DATA_BLOCK "n0016-uc164-xn10_SN50_2"   // DB1008, F_DB
{ S7_Optimized_Access := 'TRUE' }
VERSION : 0.1
// stored: InstanceOfName 00_Push-Button_Input
"00_Push-Button_Input"
BEGIN
END_DATA_BLOCK

DATA_BLOCK "n0020-uc15-el001-k30001_SN50_1"   // DB1009, F_DB
{ S7_Optimized_Access := 'TRUE' }
VERSION : 0.1
// stored: InstanceOfName 00_Push-Button_Input
"00_Push-Button_Input"
BEGIN
END_DATA_BLOCK

DATA_BLOCK "n0020-uc15-el001-k30001_SN50_2"   // DB1010, F_DB
{ S7_Optimized_Access := 'TRUE' }
VERSION : 0.1
// stored: InstanceOfName 00_Push-Button_Input
"00_Push-Button_Input"
BEGIN
END_DATA_BLOCK

DATA_BLOCK "n0020-uc15-el001-k30001_SN50_3"   // DB1011, F_DB
{ S7_Optimized_Access := 'TRUE' }
VERSION : 0.1
// stored: InstanceOfName 00_Push-Button_Input
"00_Push-Button_Input"
BEGIN
END_DATA_BLOCK

DATA_BLOCK "n0023-uc154-xn10_SN50_1"   // DB1012, F_DB
{ S7_Optimized_Access := 'TRUE' }
VERSION : 0.1
// stored: InstanceOfName 00_Push-Button_Input
"00_Push-Button_Input"
BEGIN
END_DATA_BLOCK

DATA_BLOCK "n0023-uc154-xn10_SN50_2"   // DB1013, F_DB
{ S7_Optimized_Access := 'TRUE' }
VERSION : 0.1
// stored: InstanceOfName 00_Push-Button_Input
"00_Push-Button_Input"
BEGIN
END_DATA_BLOCK

DATA_BLOCK "n0021-icg11-el001-k30001_SN50_1"   // DB1014, F_DB
{ S7_Optimized_Access := 'TRUE' }
VERSION : 0.1
// stored: InstanceOfName 00_Push-Button_Input
"00_Push-Button_Input"
BEGIN
END_DATA_BLOCK

DATA_BLOCK "n0021-icg11-el001-k30001_SN50_2"   // DB1015, F_DB
{ S7_Optimized_Access := 'TRUE' }
VERSION : 0.1
// stored: InstanceOfName 00_Push-Button_Input
"00_Push-Button_Input"
BEGIN
END_DATA_BLOCK

DATA_BLOCK "n0021-icg11-el001-k30001_SN50_3"   // DB1016, F_DB
{ S7_Optimized_Access := 'TRUE' }
VERSION : 0.1
// stored: InstanceOfName 00_Push-Button_Input
"00_Push-Button_Input"
BEGIN
END_DATA_BLOCK

DATA_BLOCK "n0021-icg11-el001-k30001_SN50_4"   // DB1017, F_DB
{ S7_Optimized_Access := 'TRUE' }
VERSION : 0.1
// stored: InstanceOfName 00_Push-Button_Input
"00_Push-Button_Input"
BEGIN
END_DATA_BLOCK

DATA_BLOCK "n0022-icg21-el001-k30001_SN50_1"   // DB1018, F_DB
{ S7_Optimized_Access := 'TRUE' }
VERSION : 0.1
// stored: InstanceOfName 00_Push-Button_Input
"00_Push-Button_Input"
BEGIN
END_DATA_BLOCK

DATA_BLOCK "n0022-icg21-el001-k30001_SN50_2"   // DB1019, F_DB
{ S7_Optimized_Access := 'TRUE' }
VERSION : 0.1
// stored: InstanceOfName 00_Push-Button_Input
"00_Push-Button_Input"
BEGIN
END_DATA_BLOCK

DATA_BLOCK "n0025-uc14-el001-k30001_SN50_1"   // DB1020, F_DB
{ S7_Optimized_Access := 'TRUE' }
VERSION : 0.1
// stored: InstanceOfName 00_Push-Button_Input
"00_Push-Button_Input"
BEGIN
END_DATA_BLOCK

DATA_BLOCK "n0025-uc14-el001-k30001_SN50_2"   // DB1021, F_DB
{ S7_Optimized_Access := 'TRUE' }
VERSION : 0.1
// stored: InstanceOfName 00_Push-Button_Input
"00_Push-Button_Input"
BEGIN
END_DATA_BLOCK

DATA_BLOCK "n0025-uc14-el001-k30001_SN50_3"   // DB1022, F_DB
{ S7_Optimized_Access := 'TRUE' }
VERSION : 0.1
// stored: InstanceOfName 00_Push-Button_Input
"00_Push-Button_Input"
BEGIN
END_DATA_BLOCK

DATA_BLOCK "n0026-uc144-xn10_SN50_1"   // DB1023, F_DB
{ S7_Optimized_Access := 'TRUE' }
VERSION : 0.1
// stored: InstanceOfName 00_Push-Button_Input
"00_Push-Button_Input"
BEGIN
END_DATA_BLOCK

DATA_BLOCK "n0026-uc144-xn10_SN50_2"   // DB1024, F_DB
{ S7_Optimized_Access := 'TRUE' }
VERSION : 0.1
// stored: InstanceOfName 00_Push-Button_Input
"00_Push-Button_Input"
BEGIN
END_DATA_BLOCK

DATA_BLOCK "n0038-uc1-el001-k30001_SN50_1"   // DB1025, F_DB
{ S7_Optimized_Access := 'TRUE' }
VERSION : 0.1
// stored: InstanceOfName 00_Push-Button_Input
"00_Push-Button_Input"
BEGIN
END_DATA_BLOCK

DATA_BLOCK "n0041-uf31-el002-k30001_SN50_1"   // DB1026, F_DB
{ S7_Optimized_Access := 'TRUE' }
VERSION : 0.1
// stored: InstanceOfName 00_Push-Button_Input
"00_Push-Button_Input"
BEGIN
END_DATA_BLOCK

DATA_BLOCK "n0044-ct1-el001-k30001_SN50_1"   // DB1027, F_DB
{ S7_Optimized_Access := 'TRUE' }
VERSION : 0.1
// stored: InstanceOfName 00_Push-Button_Input
"00_Push-Button_Input"
BEGIN
END_DATA_BLOCK

DATA_BLOCK "n0044-ct1-el001-k30001_SN50_2"   // DB1028, F_DB
{ S7_Optimized_Access := 'TRUE' }
VERSION : 0.1
// stored: InstanceOfName 00_Push-Button_Input
"00_Push-Button_Input"
BEGIN
END_DATA_BLOCK

DATA_BLOCK "n0044-ct1-el001-k30001_SN50_3"   // DB1029, F_DB
{ S7_Optimized_Access := 'TRUE' }
VERSION : 0.1
// stored: InstanceOfName 00_Push-Button_Input
"00_Push-Button_Input"
BEGIN
END_DATA_BLOCK

DATA_BLOCK "n0044-ct1-el001-k30001_SN50_4"   // DB1030, F_DB
{ S7_Optimized_Access := 'TRUE' }
VERSION : 0.1
// stored: InstanceOfName 00_Push-Button_Input
"00_Push-Button_Input"
BEGIN
END_DATA_BLOCK

DATA_BLOCK "n0045-ct1-el002-k30001_SN50_1"   // DB1031, F_DB
{ S7_Optimized_Access := 'TRUE' }
VERSION : 0.1
// stored: InstanceOfName 00_Push-Button_Input
"00_Push-Button_Input"
BEGIN
END_DATA_BLOCK

DATA_BLOCK "n0045-ct1-el002-k30001_SN50_2"   // DB1032, F_DB
{ S7_Optimized_Access := 'TRUE' }
VERSION : 0.1
// stored: InstanceOfName 00_Push-Button_Input
"00_Push-Button_Input"
BEGIN
END_DATA_BLOCK

DATA_BLOCK "n0045-ct1-el002-k30001_SN50_3"   // DB1033, F_DB
{ S7_Optimized_Access := 'TRUE' }
VERSION : 0.1
// stored: InstanceOfName 00_Push-Button_Input
"00_Push-Button_Input"
BEGIN
END_DATA_BLOCK

DATA_BLOCK "n0045-ct1-el002-k30001_SN50_4"   // DB1034, F_DB
{ S7_Optimized_Access := 'TRUE' }
VERSION : 0.1
// stored: InstanceOfName 00_Push-Button_Input
"00_Push-Button_Input"
BEGIN
END_DATA_BLOCK

DATA_BLOCK "n0045-ct1-el002-k30001_SN50_5"   // DB1035, F_DB
{ S7_Optimized_Access := 'TRUE' }
VERSION : 0.1
// stored: InstanceOfName 00_Push-Button_Input
"00_Push-Button_Input"
BEGIN
END_DATA_BLOCK

DATA_BLOCK "n0046-ct1-el003-k30001_SN50_1"   // DB1036, F_DB
{ S7_Optimized_Access := 'TRUE' }
VERSION : 0.1
// stored: InstanceOfName 00_Push-Button_Input
"00_Push-Button_Input"
BEGIN
END_DATA_BLOCK

DATA_BLOCK "n0046-ct1-el003-k30001_SN50_2"   // DB1037, F_DB
{ S7_Optimized_Access := 'TRUE' }
VERSION : 0.1
// stored: InstanceOfName 00_Push-Button_Input
"00_Push-Button_Input"
BEGIN
END_DATA_BLOCK

DATA_BLOCK "n0046-ct1-el003-k30001_SN50_3"   // DB1038, F_DB
{ S7_Optimized_Access := 'TRUE' }
VERSION : 0.1
// stored: InstanceOfName 00_Push-Button_Input
"00_Push-Button_Input"
BEGIN
END_DATA_BLOCK

DATA_BLOCK "n0046-ct1-el003-k30001_SN50_4"   // DB1039, F_DB
{ S7_Optimized_Access := 'TRUE' }
VERSION : 0.1
// stored: InstanceOfName 00_Push-Button_Input
"00_Push-Button_Input"
BEGIN
END_DATA_BLOCK

DATA_BLOCK "n0050-uc13-el001-k30001_SN50_1"   // DB1040, F_DB
{ S7_Optimized_Access := 'TRUE' }
VERSION : 0.1
// stored: InstanceOfName 00_Push-Button_Input
"00_Push-Button_Input"
BEGIN
END_DATA_BLOCK

DATA_BLOCK "n0050-uc13-el001-k30001_SN50_2"   // DB1041, F_DB
{ S7_Optimized_Access := 'TRUE' }
VERSION : 0.1
// stored: InstanceOfName 00_Push-Button_Input
"00_Push-Button_Input"
BEGIN
END_DATA_BLOCK

DATA_BLOCK "n0050-uc13-el001-k30001_SN50_3"   // DB1042, F_DB
{ S7_Optimized_Access := 'TRUE' }
VERSION : 0.1
// stored: InstanceOfName 00_Push-Button_Input
"00_Push-Button_Input"
BEGIN
END_DATA_BLOCK

DATA_BLOCK "n0051-uc134-xn10_SN50_1"   // DB1043, F_DB
{ S7_Optimized_Access := 'TRUE' }
VERSION : 0.1
// stored: InstanceOfName 00_Push-Button_Input
"00_Push-Button_Input"
BEGIN
END_DATA_BLOCK

DATA_BLOCK "n0051-uc134-xn10_SN50_2"   // DB1044, F_DB
{ S7_Optimized_Access := 'TRUE' }
VERSION : 0.1
// stored: InstanceOfName 00_Push-Button_Input
"00_Push-Button_Input"
BEGIN
END_DATA_BLOCK

DATA_BLOCK "n0053-uc12-el001-k30001_SN50_1"   // DB1045, F_DB
{ S7_Optimized_Access := 'TRUE' }
VERSION : 0.1
// stored: InstanceOfName 00_Push-Button_Input
"00_Push-Button_Input"
BEGIN
END_DATA_BLOCK

DATA_BLOCK "n0053-uc12-el001-k30001_SN50_2"   // DB1046, F_DB
{ S7_Optimized_Access := 'TRUE' }
VERSION : 0.1
// stored: InstanceOfName 00_Push-Button_Input
"00_Push-Button_Input"
BEGIN
END_DATA_BLOCK

DATA_BLOCK "n0053-uc12-el001-k30001_SN50_3"   // DB1047, F_DB
{ S7_Optimized_Access := 'TRUE' }
VERSION : 0.1
// stored: InstanceOfName 00_Push-Button_Input
"00_Push-Button_Input"
BEGIN
END_DATA_BLOCK

DATA_BLOCK "n0055-uc124-xn10_SN50_1"   // DB1048, F_DB
{ S7_Optimized_Access := 'TRUE' }
VERSION : 0.1
// stored: InstanceOfName 00_Push-Button_Input
"00_Push-Button_Input"
BEGIN
END_DATA_BLOCK

DATA_BLOCK "n0055-uc124-xn10_SN50_2"   // DB1049, F_DB
{ S7_Optimized_Access := 'TRUE' }
VERSION : 0.1
// stored: InstanceOfName 00_Push-Button_Input
"00_Push-Button_Input"
BEGIN
END_DATA_BLOCK

DATA_BLOCK "n0057-uc11-el001-k30001_SN50_1"   // DB1050, F_DB
{ S7_Optimized_Access := 'TRUE' }
VERSION : 0.1
// stored: InstanceOfName 00_Push-Button_Input
"00_Push-Button_Input"
BEGIN
END_DATA_BLOCK

DATA_BLOCK "n0057-uc11-el001-k30001_SN50_2"   // DB1051, F_DB
{ S7_Optimized_Access := 'TRUE' }
VERSION : 0.1
// stored: InstanceOfName 00_Push-Button_Input
"00_Push-Button_Input"
BEGIN
END_DATA_BLOCK

DATA_BLOCK "n0057-uc11-el001-k30001_SN50_3"   // DB1052, F_DB
{ S7_Optimized_Access := 'TRUE' }
VERSION : 0.1
// stored: InstanceOfName 00_Push-Button_Input
"00_Push-Button_Input"
BEGIN
END_DATA_BLOCK

DATA_BLOCK "n0060-uc114-xn10_SN50_1"   // DB1053, F_DB
{ S7_Optimized_Access := 'TRUE' }
VERSION : 0.1
// stored: InstanceOfName 00_Push-Button_Input
"00_Push-Button_Input"
BEGIN
END_DATA_BLOCK

DATA_BLOCK "n0060-uc114-xn10_SN50_2"   // DB1054, F_DB
{ S7_Optimized_Access := 'TRUE' }
VERSION : 0.1
// stored: InstanceOfName 00_Push-Button_Input
"00_Push-Button_Input"
BEGIN
END_DATA_BLOCK

DATA_BLOCK "n0028-uc17-el001-k30001_SN50_1"   // DB1055, F_DB
{ S7_Optimized_Access := 'TRUE' }
VERSION : 0.1
// stored: InstanceOfName 00_Push-Button_Input
"00_Push-Button_Input"
BEGIN
END_DATA_BLOCK

DATA_BLOCK "n0028-uc17-el001-k30001_SN50_2"   // DB1056, F_DB
{ S7_Optimized_Access := 'TRUE' }
VERSION : 0.1
// stored: InstanceOfName 00_Push-Button_Input
"00_Push-Button_Input"
BEGIN
END_DATA_BLOCK

DATA_BLOCK "n0029-uc173-xn10_SN50_1"   // DB1057, F_DB
{ S7_Optimized_Access := 'TRUE' }
VERSION : 0.1
// stored: InstanceOfName 00_Push-Button_Input
"00_Push-Button_Input"
BEGIN
END_DATA_BLOCK

DATA_BLOCK "n0029-uc173-xn10_SN50_2"   // DB1058, F_DB
{ S7_Optimized_Access := 'TRUE' }
VERSION : 0.1
// stored: InstanceOfName 00_Push-Button_Input
"00_Push-Button_Input"
BEGIN
END_DATA_BLOCK

DATA_BLOCK "n0033-zp001-el001-k40001_SN50_1"   // DB1059, F_DB
{ S7_Optimized_Access := 'TRUE' }
VERSION : 0.1
// stored: InstanceOfName 00_Push-Button_Input
"00_Push-Button_Input"
BEGIN
END_DATA_BLOCK

DATA_BLOCK "n0033-zp001-el001-k40001_SN50_2"   // DB1060, F_DB
{ S7_Optimized_Access := 'TRUE' }
VERSION : 0.1
// stored: InstanceOfName 00_Push-Button_Input
"00_Push-Button_Input"
BEGIN
END_DATA_BLOCK

DATA_BLOCK "n0033-zp001-el001-k40001_SN50_3"   // DB1061, F_DB
{ S7_Optimized_Access := 'TRUE' }
VERSION : 0.1
// stored: InstanceOfName 00_Push-Button_Input
"00_Push-Button_Input"
BEGIN
END_DATA_BLOCK

DATA_BLOCK "n0034-ug6-el001-k30001_SN50_1"   // DB1062, F_DB
{ S7_Optimized_Access := 'TRUE' }
VERSION : 0.1
// stored: InstanceOfName 00_Push-Button_Input
"00_Push-Button_Input"
BEGIN
END_DATA_BLOCK

DATA_BLOCK "n0034-ug6-el001-k30001_SN50_2"   // DB1063, F_DB
{ S7_Optimized_Access := 'TRUE' }
VERSION : 0.1
// stored: InstanceOfName 00_Push-Button_Input
"00_Push-Button_Input"
BEGIN
END_DATA_BLOCK

DATA_BLOCK "n0034-ug6-el001-k30001_SN50_3"   // DB1064, F_DB
{ S7_Optimized_Access := 'TRUE' }
VERSION : 0.1
// stored: InstanceOfName 00_Push-Button_Input
"00_Push-Button_Input"
BEGIN
END_DATA_BLOCK

DATA_BLOCK "n0035-ug6-xn10_SN50_1"   // DB1065, F_DB
{ S7_Optimized_Access := 'TRUE' }
VERSION : 0.1
// stored: InstanceOfName 00_Push-Button_Input
"00_Push-Button_Input"
BEGIN
END_DATA_BLOCK

DATA_BLOCK "n0035-ug6-xn10_SN50_2"   // DB1066, F_DB
{ S7_Optimized_Access := 'TRUE' }
VERSION : 0.1
// stored: InstanceOfName 00_Push-Button_Input
"00_Push-Button_Input"
BEGIN
END_DATA_BLOCK

DATA_BLOCK "n0043-db93-el001-k30001_SN50_1"   // DB1067, F_DB
{ S7_Optimized_Access := 'TRUE' }
VERSION : 0.1
// stored: InstanceOfName 00_Push-Button_Input
"00_Push-Button_Input"
BEGIN
END_DATA_BLOCK

DATA_BLOCK "n0031-db931-xn10_SN50_1"   // DB1068, F_DB
{ S7_Optimized_Access := 'TRUE' }
VERSION : 0.1
// stored: InstanceOfName 00_Push-Button_Input
"00_Push-Button_Input"
BEGIN
END_DATA_BLOCK

DATA_BLOCK "n0031-db931-xn10_SN50_2"   // DB1069, F_DB
{ S7_Optimized_Access := 'TRUE' }
VERSION : 0.1
// stored: InstanceOfName 00_Push-Button_Input
"00_Push-Button_Input"
BEGIN
END_DATA_BLOCK

DATA_BLOCK "n0005-lv008-el001-k30001_SN51_1"   // DB1070, F_DB
{ S7_Optimized_Access := 'TRUE' }
VERSION : 0.1
// stored: InstanceOfName 00_Push-Button_Input
"00_Push-Button_Input"
BEGIN
END_DATA_BLOCK

DATA_BLOCK "n0006-lv008-el001-k30001_SN51_1"   // DB1071, F_DB
{ S7_Optimized_Access := 'TRUE' }
VERSION : 0.1
// stored: InstanceOfName 00_Push-Button_Input
"00_Push-Button_Input"
BEGIN
END_DATA_BLOCK

DATA_BLOCK "n0007-icg22-el001-k30001_SN51_1"   // DB1072, F_DB
{ S7_Optimized_Access := 'TRUE' }
VERSION : 0.1
// stored: InstanceOfName 00_Push-Button_Input
"00_Push-Button_Input"
BEGIN
END_DATA_BLOCK

DATA_BLOCK "n0007-icg22-el001-k30001_SN51_2"   // DB1073, F_DB
{ S7_Optimized_Access := 'TRUE' }
VERSION : 0.1
// stored: InstanceOfName 00_Push-Button_Input
"00_Push-Button_Input"
BEGIN
END_DATA_BLOCK

DATA_BLOCK "n0008-icg12-el001-k30001_SN51_1"   // DB1074, F_DB
{ S7_Optimized_Access := 'TRUE' }
VERSION : 0.1
// stored: InstanceOfName 00_Push-Button_Input
"00_Push-Button_Input"
BEGIN
END_DATA_BLOCK

DATA_BLOCK "n0008-icg12-el001-k30001_SN51_2"   // DB1075, F_DB
{ S7_Optimized_Access := 'TRUE' }
VERSION : 0.1
// stored: InstanceOfName 00_Push-Button_Input
"00_Push-Button_Input"
BEGIN
END_DATA_BLOCK

DATA_BLOCK "n0008-icg12-el001-k30001_SN51_3"   // DB1076, F_DB
{ S7_Optimized_Access := 'TRUE' }
VERSION : 0.1
// stored: InstanceOfName 00_Push-Button_Input
"00_Push-Button_Input"
BEGIN
END_DATA_BLOCK

DATA_BLOCK "n0008-icg12-el001-k30001_SN51_4"   // DB1077, F_DB
{ S7_Optimized_Access := 'TRUE' }
VERSION : 0.1
// stored: InstanceOfName 00_Push-Button_Input
"00_Push-Button_Input"
BEGIN
END_DATA_BLOCK

DATA_BLOCK "n0026-uc915-xn10_SN51_1"   // DB1078, F_DB
{ S7_Optimized_Access := 'TRUE' }
VERSION : 0.1
// stored: InstanceOfName 00_Push-Button_Input
"00_Push-Button_Input"
BEGIN
END_DATA_BLOCK

DATA_BLOCK "n0026-uc915-xn10_SN51_2"   // DB1079, F_DB
{ S7_Optimized_Access := 'TRUE' }
VERSION : 0.1
// stored: InstanceOfName 00_Push-Button_Input
"00_Push-Button_Input"
BEGIN
END_DATA_BLOCK

DATA_BLOCK "n0027-uc915-xn11_SN51_1"   // DB1080, F_DB
{ S7_Optimized_Access := 'TRUE' }
VERSION : 0.1
// stored: InstanceOfName 00_Push-Button_Input
"00_Push-Button_Input"
BEGIN
END_DATA_BLOCK

DATA_BLOCK "n0029-ct2-el001-k30001_SN51_1"   // DB1081, F_DB
{ S7_Optimized_Access := 'TRUE' }
VERSION : 0.1
// stored: InstanceOfName 00_Push-Button_Input
"00_Push-Button_Input"
BEGIN
END_DATA_BLOCK

DATA_BLOCK "n0029-ct2-el001-k30001_SN51_2"   // DB1082, F_DB
{ S7_Optimized_Access := 'TRUE' }
VERSION : 0.1
// stored: InstanceOfName 00_Push-Button_Input
"00_Push-Button_Input"
BEGIN
END_DATA_BLOCK

DATA_BLOCK "n0029-ct2-el001-k30001_SN51_3"   // DB1083, F_DB
{ S7_Optimized_Access := 'TRUE' }
VERSION : 0.1
// stored: InstanceOfName 00_Push-Button_Input
"00_Push-Button_Input"
BEGIN
END_DATA_BLOCK

DATA_BLOCK "n0029-ct2-el001-k30001_SN51_4"   // DB1084, F_DB
{ S7_Optimized_Access := 'TRUE' }
VERSION : 0.1
// stored: InstanceOfName 00_Push-Button_Input
"00_Push-Button_Input"
BEGIN
END_DATA_BLOCK

DATA_BLOCK "n0029-ct2-el001-k30001_SN51_5"   // DB1085, F_DB
{ S7_Optimized_Access := 'TRUE' }
VERSION : 0.1
// stored: InstanceOfName 00_Push-Button_Input
"00_Push-Button_Input"
BEGIN
END_DATA_BLOCK

DATA_BLOCK "n0033-uc26-el001-k30001_SN51_1"   // DB1086, F_DB
{ S7_Optimized_Access := 'TRUE' }
VERSION : 0.1
// stored: InstanceOfName 00_Push-Button_Input
"00_Push-Button_Input"
BEGIN
END_DATA_BLOCK

DATA_BLOCK "n0033-uc26-el001-k30001_SN51_2"   // DB1087, F_DB
{ S7_Optimized_Access := 'TRUE' }
VERSION : 0.1
// stored: InstanceOfName 00_Push-Button_Input
"00_Push-Button_Input"
BEGIN
END_DATA_BLOCK

DATA_BLOCK "n0033-uc26-el001-k30001_SN51_3"   // DB1088, F_DB
{ S7_Optimized_Access := 'TRUE' }
VERSION : 0.1
// stored: InstanceOfName 00_Push-Button_Input
"00_Push-Button_Input"
BEGIN
END_DATA_BLOCK

DATA_BLOCK "n0034-uc264-xn10_SN51_1"   // DB1089, F_DB
{ S7_Optimized_Access := 'TRUE' }
VERSION : 0.1
// stored: InstanceOfName 00_Push-Button_Input
"00_Push-Button_Input"
BEGIN
END_DATA_BLOCK

DATA_BLOCK "n0034-uc264-xn10_SN51_2"   // DB1090, F_DB
{ S7_Optimized_Access := 'TRUE' }
VERSION : 0.1
// stored: InstanceOfName 00_Push-Button_Input
"00_Push-Button_Input"
BEGIN
END_DATA_BLOCK

DATA_BLOCK "n0035-ct2-el002-k30001_SN51_1"   // DB1091, F_DB
{ S7_Optimized_Access := 'TRUE' }
VERSION : 0.1
// stored: InstanceOfName 00_Push-Button_Input
"00_Push-Button_Input"
BEGIN
END_DATA_BLOCK

DATA_BLOCK "n0035-ct2-el002-k30001_SN51_2"   // DB1092, F_DB
{ S7_Optimized_Access := 'TRUE' }
VERSION : 0.1
// stored: InstanceOfName 00_Push-Button_Input
"00_Push-Button_Input"
BEGIN
END_DATA_BLOCK

DATA_BLOCK "n0035-ct2-el002-k30001_SN51_3"   // DB1093, F_DB
{ S7_Optimized_Access := 'TRUE' }
VERSION : 0.1
// stored: InstanceOfName 00_Push-Button_Input
"00_Push-Button_Input"
BEGIN
END_DATA_BLOCK

DATA_BLOCK "n0035-ct2-el002-k30001_SN51_4"   // DB1094, F_DB
{ S7_Optimized_Access := 'TRUE' }
VERSION : 0.1
// stored: InstanceOfName 00_Push-Button_Input
"00_Push-Button_Input"
BEGIN
END_DATA_BLOCK

DATA_BLOCK "n0035-ct2-el002-k30001_SN51_5"   // DB1095, F_DB
{ S7_Optimized_Access := 'TRUE' }
VERSION : 0.1
// stored: InstanceOfName 00_Push-Button_Input
"00_Push-Button_Input"
BEGIN
END_DATA_BLOCK

DATA_BLOCK "n0041-uc27-el001-k30001_SN51_1"   // DB1096, F_DB
{ S7_Optimized_Access := 'TRUE' }
VERSION : 0.1
// stored: InstanceOfName 00_Push-Button_Input
"00_Push-Button_Input"
BEGIN
END_DATA_BLOCK

DATA_BLOCK "n0041-uc27-el001-k30001_SN51_2"   // DB1097, F_DB
{ S7_Optimized_Access := 'TRUE' }
VERSION : 0.1
// stored: InstanceOfName 00_Push-Button_Input
"00_Push-Button_Input"
BEGIN
END_DATA_BLOCK

DATA_BLOCK "n0042-uc274-xn10_SN51_1"   // DB1098, F_DB
{ S7_Optimized_Access := 'TRUE' }
VERSION : 0.1
// stored: InstanceOfName 00_Push-Button_Input
"00_Push-Button_Input"
BEGIN
END_DATA_BLOCK

DATA_BLOCK "n0042-uc274-xn10_SN51_2"   // DB1099, F_DB
{ S7_Optimized_Access := 'TRUE' }
VERSION : 0.1
// stored: InstanceOfName 00_Push-Button_Input
"00_Push-Button_Input"
BEGIN
END_DATA_BLOCK

DATA_BLOCK "n0046-uc25-el001-k30001_SN51_1"   // DB1100, F_DB
{ S7_Optimized_Access := 'TRUE' }
VERSION : 0.1
// stored: InstanceOfName 00_Push-Button_Input
"00_Push-Button_Input"
BEGIN
END_DATA_BLOCK

DATA_BLOCK "n0046-uc25-el001-k30001_SN51_2"   // DB1101, F_DB
{ S7_Optimized_Access := 'TRUE' }
VERSION : 0.1
// stored: InstanceOfName 00_Push-Button_Input
"00_Push-Button_Input"
BEGIN
END_DATA_BLOCK

DATA_BLOCK "n0046-uc25-el001-k30001_SN51_3"   // DB1102, F_DB
{ S7_Optimized_Access := 'TRUE' }
VERSION : 0.1
// stored: InstanceOfName 00_Push-Button_Input
"00_Push-Button_Input"
BEGIN
END_DATA_BLOCK

DATA_BLOCK "n0047-uc254-xn10_SN51_1"   // DB1103, F_DB
{ S7_Optimized_Access := 'TRUE' }
VERSION : 0.1
// stored: InstanceOfName 00_Push-Button_Input
"00_Push-Button_Input"
BEGIN
END_DATA_BLOCK

DATA_BLOCK "n0047-uc254-xn10_SN51_2"   // DB1104, F_DB
{ S7_Optimized_Access := 'TRUE' }
VERSION : 0.1
// stored: InstanceOfName 00_Push-Button_Input
"00_Push-Button_Input"
BEGIN
END_DATA_BLOCK

DATA_BLOCK "n0051-uc24-el001-k30001_SN51_1"   // DB1105, F_DB
{ S7_Optimized_Access := 'TRUE' }
VERSION : 0.1
// stored: InstanceOfName 00_Push-Button_Input
"00_Push-Button_Input"
BEGIN
END_DATA_BLOCK

DATA_BLOCK "n0051-uc24-el001-k30001_SN51_2"   // DB1106, F_DB
{ S7_Optimized_Access := 'TRUE' }
VERSION : 0.1
// stored: InstanceOfName 00_Push-Button_Input
"00_Push-Button_Input"
BEGIN
END_DATA_BLOCK

DATA_BLOCK "n0051-uc24-el001-k30001_SN51_3"   // DB1107, F_DB
{ S7_Optimized_Access := 'TRUE' }
VERSION : 0.1
// stored: InstanceOfName 00_Push-Button_Input
"00_Push-Button_Input"
BEGIN
END_DATA_BLOCK

DATA_BLOCK "n0052-uc244-xn10_SN51_1"   // DB1108, F_DB
{ S7_Optimized_Access := 'TRUE' }
VERSION : 0.1
// stored: InstanceOfName 00_Push-Button_Input
"00_Push-Button_Input"
BEGIN
END_DATA_BLOCK

DATA_BLOCK "n0052-uc244-xn10_SN51_2"   // DB1109, F_DB
{ S7_Optimized_Access := 'TRUE' }
VERSION : 0.1
// stored: InstanceOfName 00_Push-Button_Input
"00_Push-Button_Input"
BEGIN
END_DATA_BLOCK

DATA_BLOCK "n0056-uc23-el001-k30001_SN51_1"   // DB1110, F_DB
{ S7_Optimized_Access := 'TRUE' }
VERSION : 0.1
// stored: InstanceOfName 00_Push-Button_Input
"00_Push-Button_Input"
BEGIN
END_DATA_BLOCK

DATA_BLOCK "n0056-uc23-el001-k30001_SN51_2"   // DB1111, F_DB
{ S7_Optimized_Access := 'TRUE' }
VERSION : 0.1
// stored: InstanceOfName 00_Push-Button_Input
"00_Push-Button_Input"
BEGIN
END_DATA_BLOCK

DATA_BLOCK "n0056-uc23-el001-k30001_SN51_3"   // DB1112, F_DB
{ S7_Optimized_Access := 'TRUE' }
VERSION : 0.1
// stored: InstanceOfName 00_Push-Button_Input
"00_Push-Button_Input"
BEGIN
END_DATA_BLOCK

DATA_BLOCK "n0057-uc234-xn10_SN51_1"   // DB1113, F_DB
{ S7_Optimized_Access := 'TRUE' }
VERSION : 0.1
// stored: InstanceOfName 00_Push-Button_Input
"00_Push-Button_Input"
BEGIN
END_DATA_BLOCK

DATA_BLOCK "n0057-uc234-xn10_SN51_2"   // DB1114, F_DB
{ S7_Optimized_Access := 'TRUE' }
VERSION : 0.1
// stored: InstanceOfName 00_Push-Button_Input
"00_Push-Button_Input"
BEGIN
END_DATA_BLOCK

DATA_BLOCK "n0058-ct2-el003-k30001_SN51_1"   // DB1115, F_DB
{ S7_Optimized_Access := 'TRUE' }
VERSION : 0.1
// stored: InstanceOfName 00_Push-Button_Input
"00_Push-Button_Input"
BEGIN
END_DATA_BLOCK

DATA_BLOCK "n0058-ct2-el003-k30001_SN51_2"   // DB1116, F_DB
{ S7_Optimized_Access := 'TRUE' }
VERSION : 0.1
// stored: InstanceOfName 00_Push-Button_Input
"00_Push-Button_Input"
BEGIN
END_DATA_BLOCK

DATA_BLOCK "n0058-ct2-el003-k30001_SN51_3"   // DB1117, F_DB
{ S7_Optimized_Access := 'TRUE' }
VERSION : 0.1
// stored: InstanceOfName 00_Push-Button_Input
"00_Push-Button_Input"
BEGIN
END_DATA_BLOCK

DATA_BLOCK "n0058-ct2-el003-k30001_SN51_4"   // DB1118, F_DB
{ S7_Optimized_Access := 'TRUE' }
VERSION : 0.1
// stored: InstanceOfName 00_Push-Button_Input
"00_Push-Button_Input"
BEGIN
END_DATA_BLOCK

DATA_BLOCK "n0058-ct2-el003-k30001_SN51_5"   // DB1119, F_DB
{ S7_Optimized_Access := 'TRUE' }
VERSION : 0.1
// stored: InstanceOfName 00_Push-Button_Input
"00_Push-Button_Input"
BEGIN
END_DATA_BLOCK

DATA_BLOCK "n0061-uc22-el001-k30001_SN51_1"   // DB1120, F_DB
{ S7_Optimized_Access := 'TRUE' }
VERSION : 0.1
// stored: InstanceOfName 00_Push-Button_Input
"00_Push-Button_Input"
BEGIN
END_DATA_BLOCK

DATA_BLOCK "n0061-uc22-el001-k30001_SN51_2"   // DB1121, F_DB
{ S7_Optimized_Access := 'TRUE' }
VERSION : 0.1
// stored: InstanceOfName 00_Push-Button_Input
"00_Push-Button_Input"
BEGIN
END_DATA_BLOCK

DATA_BLOCK "n0061-uc22-el001-k30001_SN51_3"   // DB1122, F_DB
{ S7_Optimized_Access := 'TRUE' }
VERSION : 0.1
// stored: InstanceOfName 00_Push-Button_Input
"00_Push-Button_Input"
BEGIN
END_DATA_BLOCK

DATA_BLOCK "n0061-uc22-el001-k30001_SN51_4"   // DB1123, F_DB
{ S7_Optimized_Access := 'TRUE' }
VERSION : 0.1
// stored: InstanceOfName 00_Push-Button_Input
"00_Push-Button_Input"
BEGIN
END_DATA_BLOCK

DATA_BLOCK "n0057-uc224-xn10_SN51_1"   // DB1124, F_DB
{ S7_Optimized_Access := 'TRUE' }
VERSION : 0.1
// stored: InstanceOfName 00_Push-Button_Input
"00_Push-Button_Input"
BEGIN
END_DATA_BLOCK

DATA_BLOCK "n0057-uc224-xn10_SN51_2"   // DB1125, F_DB
{ S7_Optimized_Access := 'TRUE' }
VERSION : 0.1
// stored: InstanceOfName 00_Push-Button_Input
"00_Push-Button_Input"
BEGIN
END_DATA_BLOCK

DATA_BLOCK "n0066-uc21-el001-k30001_SN51_1"   // DB1126, F_DB
{ S7_Optimized_Access := 'TRUE' }
VERSION : 0.1
// stored: InstanceOfName 00_Push-Button_Input
"00_Push-Button_Input"
BEGIN
END_DATA_BLOCK

DATA_BLOCK "n0066-uc21-el001-k30001_SN51_2"   // DB1127, F_DB
{ S7_Optimized_Access := 'TRUE' }
VERSION : 0.1
// stored: InstanceOfName 00_Push-Button_Input
"00_Push-Button_Input"
BEGIN
END_DATA_BLOCK

DATA_BLOCK "n0066-uc21-el001-k30001_SN51_3"   // DB1128, F_DB
{ S7_Optimized_Access := 'TRUE' }
VERSION : 0.1
// stored: InstanceOfName 00_Push-Button_Input
"00_Push-Button_Input"
BEGIN
END_DATA_BLOCK

DATA_BLOCK "n0067-uc214-xn10_SN51_1"   // DB1129, F_DB
{ S7_Optimized_Access := 'TRUE' }
VERSION : 0.1
// stored: InstanceOfName 00_Push-Button_Input
"00_Push-Button_Input"
BEGIN
END_DATA_BLOCK

DATA_BLOCK "n0067-uc214-xn10_SN51_2"   // DB1130, F_DB
{ S7_Optimized_Access := 'TRUE' }
VERSION : 0.1
// stored: InstanceOfName 00_Push-Button_Input
"00_Push-Button_Input"
BEGIN
END_DATA_BLOCK

DATA_BLOCK "n0070-uf31-el001-k30001_SN51_1"   // DB1131, F_DB
{ S7_Optimized_Access := 'TRUE' }
VERSION : 0.1
// stored: InstanceOfName 00_Push-Button_Input
"00_Push-Button_Input"
BEGIN
END_DATA_BLOCK

DATA_BLOCK "n0072-uf51-el001-k30001_SN51_1"   // DB1132, F_DB
{ S7_Optimized_Access := 'TRUE' }
VERSION : 0.1
// stored: InstanceOfName 00_Push-Button_Input
"00_Push-Button_Input"
BEGIN
END_DATA_BLOCK

DATA_BLOCK "n0080-uf511-xn10_SN51_1"   // DB1133, F_DB
{ S7_Optimized_Access := 'TRUE' }
VERSION : 0.1
// stored: InstanceOfName 00_Push-Button_Input
"00_Push-Button_Input"
BEGIN
END_DATA_BLOCK

DATA_BLOCK "n0073-ifg31-el001-k30001_SN51_1"   // DB1134, F_DB
{ S7_Optimized_Access := 'TRUE' }
VERSION : 0.1
// stored: InstanceOfName 00_Push-Button_Input
"00_Push-Button_Input"
BEGIN
END_DATA_BLOCK

DATA_BLOCK "n0073-ifg31-el001-k30001_SN51_2"   // DB1135, F_DB
{ S7_Optimized_Access := 'TRUE' }
VERSION : 0.1
// stored: InstanceOfName 00_Push-Button_Input
"00_Push-Button_Input"
BEGIN
END_DATA_BLOCK

DATA_BLOCK "n0074-ifg41-el001-k30001_SN51_1"   // DB1136, F_DB
{ S7_Optimized_Access := 'TRUE' }
VERSION : 0.1
// stored: InstanceOfName 00_Push-Button_Input
"00_Push-Button_Input"
BEGIN
END_DATA_BLOCK

DATA_BLOCK "n0075-uf32-el001-k30001_SN51_1"   // DB1137, F_DB
{ S7_Optimized_Access := 'TRUE' }
VERSION : 0.1
// stored: InstanceOfName 00_Push-Button_Input
"00_Push-Button_Input"
BEGIN
END_DATA_BLOCK

DATA_BLOCK "n0082-zp002-el001-k30001_SN51_1"   // DB1138, F_DB
{ S7_Optimized_Access := 'TRUE' }
VERSION : 0.1
// stored: InstanceOfName 00_Push-Button_Input
"00_Push-Button_Input"
BEGIN
END_DATA_BLOCK

DATA_BLOCK "n0083-lv001-el001-k30001_SN51_1"   // DB1139, F_DB
{ S7_Optimized_Access := 'TRUE' }
VERSION : 0.1
// stored: InstanceOfName 00_Push-Button_Input
"00_Push-Button_Input"
BEGIN
END_DATA_BLOCK

DATA_BLOCK "n0084-lv001-el001-k30001_SN51_1"   // DB1140, F_DB
{ S7_Optimized_Access := 'TRUE' }
VERSION : 0.1
// stored: InstanceOfName 00_Push-Button_Input
"00_Push-Button_Input"
BEGIN
END_DATA_BLOCK

DATA_BLOCK "n0085-uc29-el001-k30001_SN51_1"   // DB1141, F_DB
{ S7_Optimized_Access := 'TRUE' }
VERSION : 0.1
// stored: InstanceOfName 00_Push-Button_Input
"00_Push-Button_Input"
BEGIN
END_DATA_BLOCK

DATA_BLOCK "n0085-uc29-el001-k30001_SN51_2"   // DB1142, F_DB
{ S7_Optimized_Access := 'TRUE' }
VERSION : 0.1
// stored: InstanceOfName 00_Push-Button_Input
"00_Push-Button_Input"
BEGIN
END_DATA_BLOCK

DATA_BLOCK "n0091-zp001-el001-k30001_SN51_1"   // DB1143, F_DB
{ S7_Optimized_Access := 'TRUE' }
VERSION : 0.1
// stored: InstanceOfName 00_Push-Button_Input
"00_Push-Button_Input"
BEGIN
END_DATA_BLOCK

DATA_BLOCK "n0091-zp001-el001-k30001_SN51_2"   // DB1144, F_DB
{ S7_Optimized_Access := 'TRUE' }
VERSION : 0.1
// stored: InstanceOfName 00_Push-Button_Input
"00_Push-Button_Input"
BEGIN
END_DATA_BLOCK

DATA_BLOCK "n0093-ug7-el001-k30001_SN51_1"   // DB1145, F_DB
{ S7_Optimized_Access := 'TRUE' }
VERSION : 0.1
// stored: InstanceOfName 00_Push-Button_Input
"00_Push-Button_Input"
BEGIN
END_DATA_BLOCK

DATA_BLOCK "n0093-ug7-el001-k30001_SN51_2"   // DB1146, F_DB
{ S7_Optimized_Access := 'TRUE' }
VERSION : 0.1
// stored: InstanceOfName 00_Push-Button_Input
"00_Push-Button_Input"
BEGIN
END_DATA_BLOCK

DATA_BLOCK "n0093-ug7-el001-k30001_SN51_3"   // DB1147, F_DB
{ S7_Optimized_Access := 'TRUE' }
VERSION : 0.1
// stored: InstanceOfName 00_Push-Button_Input
"00_Push-Button_Input"
BEGIN
END_DATA_BLOCK

DATA_BLOCK "n0094-ug7-xn10_SN51_1"   // DB1148, F_DB
{ S7_Optimized_Access := 'TRUE' }
VERSION : 0.1
// stored: InstanceOfName 00_Push-Button_Input
"00_Push-Button_Input"
BEGIN
END_DATA_BLOCK

DATA_BLOCK "n0094-ug7-xn10_SN51_2"   // DB1149, F_DB
{ S7_Optimized_Access := 'TRUE' }
VERSION : 0.1
// stored: InstanceOfName 00_Push-Button_Input
"00_Push-Button_Input"
BEGIN
END_DATA_BLOCK

// folder: 01_Feedback error

DATA_BLOCK "FDBACK error_EXAMPLE"   // DB16, F_DB
{ S7_Optimized_Access := 'TRUE' }
VERSION : 0.1
// stored: InstanceOfName 03_FDBACK error
"03_FDBACK error"
BEGIN
END_DATA_BLOCK

DATA_BLOCK "FDBACK-N0001-1"   // DB19, F_DB
{ S7_Optimized_Access := 'TRUE' }
VERSION : 0.1
// stored: InstanceOfName 03_FDBACK error
"03_FDBACK error"
BEGIN
END_DATA_BLOCK

DATA_BLOCK "FDBK_Error_n0015-uc16-el001-k30001_SN50_1"   // DB2000, F_DB
{ S7_Optimized_Access := 'TRUE' }
VERSION : 0.1
// stored: InstanceOfName 03_FDBACK error
"03_FDBACK error"
BEGIN
END_DATA_BLOCK

DATA_BLOCK "FDBK_Error_n0015-uc16-el001-k30001_SN50_2"   // DB2001, F_DB
{ S7_Optimized_Access := 'TRUE' }
VERSION : 0.1
// stored: InstanceOfName 03_FDBACK error
"03_FDBACK error"
BEGIN
END_DATA_BLOCK

DATA_BLOCK "FDBK_Error_n0015-uc16-el001-k30001_SN50_3"   // DB2002, F_DB
{ S7_Optimized_Access := 'TRUE' }
VERSION : 0.1
// stored: InstanceOfName 03_FDBACK error
"03_FDBACK error"
BEGIN
END_DATA_BLOCK

DATA_BLOCK "FDBK_Error_n0017-lv004-el001-k30001_SN50_1"   // DB2003, F_DB
{ S7_Optimized_Access := 'TRUE' }
VERSION : 0.1
// stored: InstanceOfName 03_FDBACK error
"03_FDBACK error"
BEGIN
END_DATA_BLOCK

DATA_BLOCK "FDBK_Error_n0018-lv004-el001-k30001_SN50_1"   // DB2004, F_DB
{ S7_Optimized_Access := 'TRUE' }
VERSION : 0.1
// stored: InstanceOfName 03_FDBACK error
"03_FDBACK error"
BEGIN
END_DATA_BLOCK

DATA_BLOCK "FDBK_Error_n0020-uc15-el001-k30001_SN50_1"   // DB2005, F_DB
{ S7_Optimized_Access := 'TRUE' }
VERSION : 0.1
// stored: InstanceOfName 03_FDBACK error
"03_FDBACK error"
BEGIN
END_DATA_BLOCK

DATA_BLOCK "FDBK_Error_n0020-uc15-el001-k30001_SN50_2"   // DB2006, F_DB
{ S7_Optimized_Access := 'TRUE' }
VERSION : 0.1
// stored: InstanceOfName 03_FDBACK error
"03_FDBACK error"
BEGIN
END_DATA_BLOCK

DATA_BLOCK "FDBK_Error_n0020-uc15-el001-k30001_SN50_3"   // DB2007, F_DB
{ S7_Optimized_Access := 'TRUE' }
VERSION : 0.1
// stored: InstanceOfName 03_FDBACK error
"03_FDBACK error"
BEGIN
END_DATA_BLOCK

DATA_BLOCK "FDBK_Error_n0021-icg11-el001-k30001_SN50_1"   // DB2008, F_DB
{ S7_Optimized_Access := 'TRUE' }
VERSION : 0.1
// stored: InstanceOfName 03_FDBACK error
"03_FDBACK error"
BEGIN
END_DATA_BLOCK

DATA_BLOCK "FDBK_Error_n0022-icg21-el001-k30001_SN50_1"   // DB2009, F_DB
{ S7_Optimized_Access := 'TRUE' }
VERSION : 0.1
// stored: InstanceOfName 03_FDBACK error
"03_FDBACK error"
BEGIN
END_DATA_BLOCK

DATA_BLOCK "FDBK_Error_n0025-uc14-el001-k30001_SN50_1"   // DB2010, F_DB
{ S7_Optimized_Access := 'TRUE' }
VERSION : 0.1
// stored: InstanceOfName 03_FDBACK error
"03_FDBACK error"
BEGIN
END_DATA_BLOCK

DATA_BLOCK "FDBK_Error_n0025-uc14-el001-k30001_SN50_2"   // DB2011, F_DB
{ S7_Optimized_Access := 'TRUE' }
VERSION : 0.1
// stored: InstanceOfName 03_FDBACK error
"03_FDBACK error"
BEGIN
END_DATA_BLOCK

DATA_BLOCK "FDBK_Error_n0025-uc14-el001-k30001_SN50_3"   // DB2012, F_DB
{ S7_Optimized_Access := 'TRUE' }
VERSION : 0.1
// stored: InstanceOfName 03_FDBACK error
"03_FDBACK error"
BEGIN
END_DATA_BLOCK

DATA_BLOCK "FDBK_Error_n0039-lv001-el001-k30001_SN50_1"   // DB2013, F_DB
{ S7_Optimized_Access := 'TRUE' }
VERSION : 0.1
// stored: InstanceOfName 03_FDBACK error
"03_FDBACK error"
BEGIN
END_DATA_BLOCK

DATA_BLOCK "FDBK_Error_n0040-lv001-el001-k30001_SN50_1"   // DB2014, F_DB
{ S7_Optimized_Access := 'TRUE' }
VERSION : 0.1
// stored: InstanceOfName 03_FDBACK error
"03_FDBACK error"
BEGIN
END_DATA_BLOCK

DATA_BLOCK "FDBK_Error_n0041-uf31-el002-k30001_SN50_1"   // DB2015, F_DB
{ S7_Optimized_Access := 'TRUE' }
VERSION : 0.1
// stored: InstanceOfName 03_FDBACK error
"03_FDBACK error"
BEGIN
END_DATA_BLOCK

DATA_BLOCK "FDBK_Error_n0042-uf41-el002-k30001_SN50_1"   // DB2016, F_DB
{ S7_Optimized_Access := 'TRUE' }
VERSION : 0.1
// stored: InstanceOfName 03_FDBACK error
"03_FDBACK error"
BEGIN
END_DATA_BLOCK

DATA_BLOCK "FDBK_Error_n0044-ct1-el001-k30001_SN50_1"   // DB2017, F_DB
{ S7_Optimized_Access := 'TRUE' }
VERSION : 0.1
// stored: InstanceOfName 03_FDBACK error
"03_FDBACK error"
BEGIN
END_DATA_BLOCK

DATA_BLOCK "FDBK_Error_n0045-ct1-el002-k30001_SN50_1"   // DB2018, F_DB
{ S7_Optimized_Access := 'TRUE' }
VERSION : 0.1
// stored: InstanceOfName 03_FDBACK error
"03_FDBACK error"
BEGIN
END_DATA_BLOCK

DATA_BLOCK "FDBK_Error_n0046-ct1-el003-k30001_SN50_1"   // DB2019, F_DB
{ S7_Optimized_Access := 'TRUE' }
VERSION : 0.1
// stored: InstanceOfName 03_FDBACK error
"03_FDBACK error"
BEGIN
END_DATA_BLOCK

DATA_BLOCK "FDBK_Error_n0047-lv002-el001-k30001_SN50_1"   // DB2020, F_DB
{ S7_Optimized_Access := 'TRUE' }
VERSION : 0.1
// stored: InstanceOfName 03_FDBACK error
"03_FDBACK error"
BEGIN
END_DATA_BLOCK

DATA_BLOCK "FDBK_Error_n0048-lv002-el001-k30001_SN50_1"   // DB2021, F_DB
{ S7_Optimized_Access := 'TRUE' }
VERSION : 0.1
// stored: InstanceOfName 03_FDBACK error
"03_FDBACK error"
BEGIN
END_DATA_BLOCK

DATA_BLOCK "FDBK_Error_n0050-uc13-el001-k30001_SN50_1"   // DB2022, F_DB
{ S7_Optimized_Access := 'TRUE' }
VERSION : 0.1
// stored: InstanceOfName 03_FDBACK error
"03_FDBACK error"
BEGIN
END_DATA_BLOCK

DATA_BLOCK "FDBK_Error_n0050-uc13-el001-k30001_SN50_2"   // DB2023, F_DB
{ S7_Optimized_Access := 'TRUE' }
VERSION : 0.1
// stored: InstanceOfName 03_FDBACK error
"03_FDBACK error"
BEGIN
END_DATA_BLOCK

DATA_BLOCK "FDBK_Error_n0050-uc13-el001-k30001_SN50_3"   // DB2024, F_DB
{ S7_Optimized_Access := 'TRUE' }
VERSION : 0.1
// stored: InstanceOfName 03_FDBACK error
"03_FDBACK error"
BEGIN
END_DATA_BLOCK

DATA_BLOCK "FDBK_Error_n0053-uc12-el001-k30001_SN50_1"   // DB2025, F_DB
{ S7_Optimized_Access := 'TRUE' }
VERSION : 0.1
// stored: InstanceOfName 03_FDBACK error
"03_FDBACK error"
BEGIN
END_DATA_BLOCK

DATA_BLOCK "FDBK_Error_n0053-uc12-el001-k30001_SN50_2"   // DB2026, F_DB
{ S7_Optimized_Access := 'TRUE' }
VERSION : 0.1
// stored: InstanceOfName 03_FDBACK error
"03_FDBACK error"
BEGIN
END_DATA_BLOCK

DATA_BLOCK "FDBK_Error_n0053-uc12-el001-k30001_SN50_3"   // DB2027, F_DB
{ S7_Optimized_Access := 'TRUE' }
VERSION : 0.1
// stored: InstanceOfName 03_FDBACK error
"03_FDBACK error"
BEGIN
END_DATA_BLOCK

DATA_BLOCK "FDBK_Error_n0054-uf31-el003-k30001_SN50_1"   // DB2028, F_DB
{ S7_Optimized_Access := 'TRUE' }
VERSION : 0.1
// stored: InstanceOfName 03_FDBACK error
"03_FDBACK error"
BEGIN
END_DATA_BLOCK

DATA_BLOCK "FDBK_Error_n0057-uc11-el001-k30001_SN50_1"   // DB2029, F_DB
{ S7_Optimized_Access := 'TRUE' }
VERSION : 0.1
// stored: InstanceOfName 03_FDBACK error
"03_FDBACK error"
BEGIN
END_DATA_BLOCK

DATA_BLOCK "FDBK_Error_n0057-uc11-el001-k30001_SN50_2"   // DB2030, F_DB
{ S7_Optimized_Access := 'TRUE' }
VERSION : 0.1
// stored: InstanceOfName 03_FDBACK error
"03_FDBACK error"
BEGIN
END_DATA_BLOCK

DATA_BLOCK "FDBK_Error_n0057-uc11-el001-k30001_SN50_3"   // DB2031, F_DB
{ S7_Optimized_Access := 'TRUE' }
VERSION : 0.1
// stored: InstanceOfName 03_FDBACK error
"03_FDBACK error"
BEGIN
END_DATA_BLOCK

DATA_BLOCK "FDBK_Error_n0058-lv003-el001-k30001_SN50_1"   // DB2032, F_DB
{ S7_Optimized_Access := 'TRUE' }
VERSION : 0.1
// stored: InstanceOfName 03_FDBACK error
"03_FDBACK error"
BEGIN
END_DATA_BLOCK

DATA_BLOCK "FDBK_Error_n0059-lv003-el001-k30001_SN50_1"   // DB2033, F_DB
{ S7_Optimized_Access := 'TRUE' }
VERSION : 0.1
// stored: InstanceOfName 03_FDBACK error
"03_FDBACK error"
BEGIN
END_DATA_BLOCK

DATA_BLOCK "FDBK_Error_n0028-uc17-el001-k30001_SN50_1"   // DB2034, F_DB
{ S7_Optimized_Access := 'TRUE' }
VERSION : 0.1
// stored: InstanceOfName 03_FDBACK error
"03_FDBACK error"
BEGIN
END_DATA_BLOCK

DATA_BLOCK "FDBK_Error_n0028-uc17-el001-k30001_SN50_2"   // DB2035, F_DB
{ S7_Optimized_Access := 'TRUE' }
VERSION : 0.1
// stored: InstanceOfName 03_FDBACK error
"03_FDBACK error"
BEGIN
END_DATA_BLOCK

DATA_BLOCK "FDBK_Error_n0033-zp001-el001-k40001_SN50_1"   // DB2036, F_DB
{ S7_Optimized_Access := 'TRUE' }
VERSION : 0.1
// stored: InstanceOfName 03_FDBACK error
"03_FDBACK error"
BEGIN
END_DATA_BLOCK

DATA_BLOCK "FDBK_Error_n0033-zp001-el001-k40001_SN50_2"   // DB2037, F_DB
{ S7_Optimized_Access := 'TRUE' }
VERSION : 0.1
// stored: InstanceOfName 03_FDBACK error
"03_FDBACK error"
BEGIN
END_DATA_BLOCK

DATA_BLOCK "FDBK_Error_n0034-ug6-el001-k30001_SN50_1"   // DB2038, F_DB
{ S7_Optimized_Access := 'TRUE' }
VERSION : 0.1
// stored: InstanceOfName 03_FDBACK error
"03_FDBACK error"
BEGIN
END_DATA_BLOCK

DATA_BLOCK "FDBK_Error_n0034-ug6-el001-k30001_SN50_2"   // DB2039, F_DB
{ S7_Optimized_Access := 'TRUE' }
VERSION : 0.1
// stored: InstanceOfName 03_FDBACK error
"03_FDBACK error"
BEGIN
END_DATA_BLOCK

DATA_BLOCK "FDBK_Error_n0034-ug6-el001-k30001_SN50_3"   // DB2040, F_DB
{ S7_Optimized_Access := 'TRUE' }
VERSION : 0.1
// stored: InstanceOfName 03_FDBACK error
"03_FDBACK error"
BEGIN
END_DATA_BLOCK

DATA_BLOCK "FDBK_Error_n0043-db93-el001-k30001_SN50_1"   // DB2041, F_DB
{ S7_Optimized_Access := 'TRUE' }
VERSION : 0.1
// stored: InstanceOfName 03_FDBACK error
"03_FDBACK error"
BEGIN
END_DATA_BLOCK

DATA_BLOCK "FDBK_Error_n0005-lv008-el001-k30001_SN51_1"   // DB2042, F_DB
{ S7_Optimized_Access := 'TRUE' }
VERSION : 0.1
// stored: InstanceOfName 03_FDBACK error
"03_FDBACK error"
BEGIN
END_DATA_BLOCK

DATA_BLOCK "FDBK_Error_n0006-lv008-el001-k30001_SN51_1"   // DB2043, F_DB
{ S7_Optimized_Access := 'TRUE' }
VERSION : 0.1
// stored: InstanceOfName 03_FDBACK error
"03_FDBACK error"
BEGIN
END_DATA_BLOCK

DATA_BLOCK "FDBK_Error_n0007-icg22-el001-k30001_SN51_1"   // DB2044, F_DB
{ S7_Optimized_Access := 'TRUE' }
VERSION : 0.1
// stored: InstanceOfName 03_FDBACK error
"03_FDBACK error"
BEGIN
END_DATA_BLOCK

DATA_BLOCK "FDBK_Error_n0008-icg12-el001-k30001_SN51_1"   // DB2045, F_DB
{ S7_Optimized_Access := 'TRUE' }
VERSION : 0.1
// stored: InstanceOfName 03_FDBACK error
"03_FDBACK error"
BEGIN
END_DATA_BLOCK

DATA_BLOCK "FDBK_Error_n0009-uf42-el002-k30001_SN51_1"   // DB2046, F_DB
{ S7_Optimized_Access := 'TRUE' }
VERSION : 0.1
// stored: InstanceOfName 03_FDBACK error
"03_FDBACK error"
BEGIN
END_DATA_BLOCK

DATA_BLOCK "FDBK_Error_n0010-lv007-el001-k30001_SN51_1"   // DB2047, F_DB
{ S7_Optimized_Access := 'TRUE' }
VERSION : 0.1
// stored: InstanceOfName 03_FDBACK error
"03_FDBACK error"
BEGIN
END_DATA_BLOCK

DATA_BLOCK "FDBK_Error_n0011-lv007-el001-k30001_SN51_1"   // DB2048, F_DB
{ S7_Optimized_Access := 'TRUE' }
VERSION : 0.1
// stored: InstanceOfName 03_FDBACK error
"03_FDBACK error"
BEGIN
END_DATA_BLOCK

DATA_BLOCK "FDBK_Error_n0025-dc91-el001-k30001_SN51_1"   // DB2049, F_DB
{ S7_Optimized_Access := 'TRUE' }
VERSION : 0.1
// stored: InstanceOfName 03_FDBACK error
"03_FDBACK error"
BEGIN
END_DATA_BLOCK

DATA_BLOCK "FDBK_Error_n0028-lv005-el001-k30001_SN51_1"   // DB2050, F_DB
{ S7_Optimized_Access := 'TRUE' }
VERSION : 0.1
// stored: InstanceOfName 03_FDBACK error
"03_FDBACK error"
BEGIN
END_DATA_BLOCK

DATA_BLOCK "FDBK_Error_n0029-ct2-el001-k30001_SN51_1"   // DB2051, F_DB
{ S7_Optimized_Access := 'TRUE' }
VERSION : 0.1
// stored: InstanceOfName 03_FDBACK error
"03_FDBACK error"
BEGIN
END_DATA_BLOCK

DATA_BLOCK "FDBK_Error_n0033-uc26-el001-k30001_SN51_1"   // DB2052, F_DB
{ S7_Optimized_Access := 'TRUE' }
VERSION : 0.1
// stored: InstanceOfName 03_FDBACK error
"03_FDBACK error"
BEGIN
END_DATA_BLOCK

DATA_BLOCK "FDBK_Error_n0033-uc26-el001-k30001_SN51_2"   // DB2053, F_DB
{ S7_Optimized_Access := 'TRUE' }
VERSION : 0.1
// stored: InstanceOfName 03_FDBACK error
"03_FDBACK error"
BEGIN
END_DATA_BLOCK

DATA_BLOCK "FDBK_Error_n0033-uc26-el001-k30001_SN51_3"   // DB2054, F_DB
{ S7_Optimized_Access := 'TRUE' }
VERSION : 0.1
// stored: InstanceOfName 03_FDBACK error
"03_FDBACK error"
BEGIN
END_DATA_BLOCK

DATA_BLOCK "FDBK_Error_n0035-ct2-el002-k30001_SN51_1"   // DB2055, F_DB
{ S7_Optimized_Access := 'TRUE' }
VERSION : 0.1
// stored: InstanceOfName 03_FDBACK error
"03_FDBACK error"
BEGIN
END_DATA_BLOCK

DATA_BLOCK "FDBK_Error_n0036-lv005-el001-k30001_SN51_1"   // DB2056, F_DB
{ S7_Optimized_Access := 'TRUE' }
VERSION : 0.1
// stored: InstanceOfName 03_FDBACK error
"03_FDBACK error"
BEGIN
END_DATA_BLOCK

DATA_BLOCK "FDBK_Error_n0041-uc27-el001-k30001_SN51_1"   // DB2057, F_DB
{ S7_Optimized_Access := 'TRUE' }
VERSION : 0.1
// stored: InstanceOfName 03_FDBACK error
"03_FDBACK error"
BEGIN
END_DATA_BLOCK

DATA_BLOCK "FDBK_Error_n0041-uc27-el001-k30001_SN51_2"   // DB2058, F_DB
{ S7_Optimized_Access := 'TRUE' }
VERSION : 0.1
// stored: InstanceOfName 03_FDBACK error
"03_FDBACK error"
BEGIN
END_DATA_BLOCK

DATA_BLOCK "FDBK_Error_n0046-uc25-el001-k30001_SN51_1"   // DB2059, F_DB
{ S7_Optimized_Access := 'TRUE' }
VERSION : 0.1
// stored: InstanceOfName 03_FDBACK error
"03_FDBACK error"
BEGIN
END_DATA_BLOCK

DATA_BLOCK "FDBK_Error_n0046-uc25-el001-k30001_SN51_2"   // DB2060, F_DB
{ S7_Optimized_Access := 'TRUE' }
VERSION : 0.1
// stored: InstanceOfName 03_FDBACK error
"03_FDBACK error"
BEGIN
END_DATA_BLOCK

DATA_BLOCK "FDBK_Error_n0046-uc25-el001-k30001_SN51_3"   // DB2061, F_DB
{ S7_Optimized_Access := 'TRUE' }
VERSION : 0.1
// stored: InstanceOfName 03_FDBACK error
"03_FDBACK error"
BEGIN
END_DATA_BLOCK

DATA_BLOCK "FDBK_Error_n0048-lv006-el001-k30001_SN51_1"   // DB2062, F_DB
{ S7_Optimized_Access := 'TRUE' }
VERSION : 0.1
// stored: InstanceOfName 03_FDBACK error
"03_FDBACK error"
BEGIN
END_DATA_BLOCK

DATA_BLOCK "FDBK_Error_n0051-uc24-el001-k30001_SN51_1"   // DB2063, F_DB
{ S7_Optimized_Access := 'TRUE' }
VERSION : 0.1
// stored: InstanceOfName 03_FDBACK error
"03_FDBACK error"
BEGIN
END_DATA_BLOCK

DATA_BLOCK "FDBK_Error_n0051-uc24-el001-k30001_SN51_2"   // DB2064, F_DB
{ S7_Optimized_Access := 'TRUE' }
VERSION : 0.1
// stored: InstanceOfName 03_FDBACK error
"03_FDBACK error"
BEGIN
END_DATA_BLOCK

DATA_BLOCK "FDBK_Error_n0051-uc24-el001-k30001_SN51_3"   // DB2065, F_DB
{ S7_Optimized_Access := 'TRUE' }
VERSION : 0.1
// stored: InstanceOfName 03_FDBACK error
"03_FDBACK error"
BEGIN
END_DATA_BLOCK

DATA_BLOCK "FDBK_Error_n0056-uc23-el001-k30001_SN51_1"   // DB2066, F_DB
{ S7_Optimized_Access := 'TRUE' }
VERSION : 0.1
// stored: InstanceOfName 03_FDBACK error
"03_FDBACK error"
BEGIN
END_DATA_BLOCK

DATA_BLOCK "FDBK_Error_n0056-uc23-el001-k30001_SN51_2"   // DB2067, F_DB
{ S7_Optimized_Access := 'TRUE' }
VERSION : 0.1
// stored: InstanceOfName 03_FDBACK error
"03_FDBACK error"
BEGIN
END_DATA_BLOCK

DATA_BLOCK "FDBK_Error_n0056-uc23-el001-k30001_SN51_3"   // DB2068, F_DB
{ S7_Optimized_Access := 'TRUE' }
VERSION : 0.1
// stored: InstanceOfName 03_FDBACK error
"03_FDBACK error"
BEGIN
END_DATA_BLOCK

DATA_BLOCK "FDBK_Error_n0058-ct2-el003-k30001_SN51_1"   // DB2069, F_DB
{ S7_Optimized_Access := 'TRUE' }
VERSION : 0.1
// stored: InstanceOfName 03_FDBACK error
"03_FDBACK error"
BEGIN
END_DATA_BLOCK

DATA_BLOCK "FDBK_Error_n0061-uc22-el001-k30001_SN51_1"   // DB2070, F_DB
{ S7_Optimized_Access := 'TRUE' }
VERSION : 0.1
// stored: InstanceOfName 03_FDBACK error
"03_FDBACK error"
BEGIN
END_DATA_BLOCK

DATA_BLOCK "FDBK_Error_n0061-uc22-el001-k30001_SN51_2"   // DB2071, F_DB
{ S7_Optimized_Access := 'TRUE' }
VERSION : 0.1
// stored: InstanceOfName 03_FDBACK error
"03_FDBACK error"
BEGIN
END_DATA_BLOCK

DATA_BLOCK "FDBK_Error_n0061-uc22-el001-k30001_SN51_3"   // DB2072, F_DB
{ S7_Optimized_Access := 'TRUE' }
VERSION : 0.1
// stored: InstanceOfName 03_FDBACK error
"03_FDBACK error"
BEGIN
END_DATA_BLOCK

DATA_BLOCK "FDBK_Error_n0063-lv006-el001-k30001_SN51_1"   // DB2073, F_DB
{ S7_Optimized_Access := 'TRUE' }
VERSION : 0.1
// stored: InstanceOfName 03_FDBACK error
"03_FDBACK error"
BEGIN
END_DATA_BLOCK

DATA_BLOCK "FDBK_Error_n0066-uc21-el001-k30001_SN51_1"   // DB2074, F_DB
{ S7_Optimized_Access := 'TRUE' }
VERSION : 0.1
// stored: InstanceOfName 03_FDBACK error
"03_FDBACK error"
BEGIN
END_DATA_BLOCK

DATA_BLOCK "FDBK_Error_n0066-uc21-el001-k30001_SN51_2"   // DB2075, F_DB
{ S7_Optimized_Access := 'TRUE' }
VERSION : 0.1
// stored: InstanceOfName 03_FDBACK error
"03_FDBACK error"
BEGIN
END_DATA_BLOCK

DATA_BLOCK "FDBK_Error_n0066-uc21-el001-k30001_SN51_3"   // DB2076, F_DB
{ S7_Optimized_Access := 'TRUE' }
VERSION : 0.1
// stored: InstanceOfName 03_FDBACK error
"03_FDBACK error"
BEGIN
END_DATA_BLOCK

DATA_BLOCK "FDBK_Error_n0070-uf31-el001-k30001_SN51_1"   // DB2077, F_DB
{ S7_Optimized_Access := 'TRUE' }
VERSION : 0.1
// stored: InstanceOfName 03_FDBACK error
"03_FDBACK error"
BEGIN
END_DATA_BLOCK

DATA_BLOCK "FDBK_Error_n0071-uf41-el001-k30001_SN51_1"   // DB2078, F_DB
{ S7_Optimized_Access := 'TRUE' }
VERSION : 0.1
// stored: InstanceOfName 03_FDBACK error
"03_FDBACK error"
BEGIN
END_DATA_BLOCK

DATA_BLOCK "FDBK_Error_n0072-uf51-el001-k30001_SN51_1"   // DB2079, F_DB
{ S7_Optimized_Access := 'TRUE' }
VERSION : 0.1
// stored: InstanceOfName 03_FDBACK error
"03_FDBACK error"
BEGIN
END_DATA_BLOCK

DATA_BLOCK "FDBK_Error_n0073-ifg31-el001-k30001_SN51_1"   // DB2080, F_DB
{ S7_Optimized_Access := 'TRUE' }
VERSION : 0.1
// stored: InstanceOfName 03_FDBACK error
"03_FDBACK error"
BEGIN
END_DATA_BLOCK

DATA_BLOCK "FDBK_Error_n0074-ifg41-el001-k30001_SN51_1"   // DB2081, F_DB
{ S7_Optimized_Access := 'TRUE' }
VERSION : 0.1
// stored: InstanceOfName 03_FDBACK error
"03_FDBACK error"
BEGIN
END_DATA_BLOCK

DATA_BLOCK "FDBK_Error_n0075-uf32-el001-k30001_SN51_1"   // DB2082, F_DB
{ S7_Optimized_Access := 'TRUE' }
VERSION : 0.1
// stored: InstanceOfName 03_FDBACK error
"03_FDBACK error"
BEGIN
END_DATA_BLOCK

DATA_BLOCK "FDBK_Error_n0076-uf42-el001-k30001_SN51_1"   // DB2083, F_DB
{ S7_Optimized_Access := 'TRUE' }
VERSION : 0.1
// stored: InstanceOfName 03_FDBACK error
"03_FDBACK error"
BEGIN
END_DATA_BLOCK

DATA_BLOCK "FDBK_Error_n0082-zp002-el001-k30001_SN51_1"   // DB2084, F_DB
{ S7_Optimized_Access := 'TRUE' }
VERSION : 0.1
// stored: InstanceOfName 03_FDBACK error
"03_FDBACK error"
BEGIN
END_DATA_BLOCK

DATA_BLOCK "FDBK_Error_n0083-lv001-el001-k30001_SN51_1"   // DB2085, F_DB
{ S7_Optimized_Access := 'TRUE' }
VERSION : 0.1
// stored: InstanceOfName 03_FDBACK error
"03_FDBACK error"
BEGIN
END_DATA_BLOCK

DATA_BLOCK "FDBK_Error_n0084-lv001-el001-k30001_SN51_1"   // DB2086, F_DB
{ S7_Optimized_Access := 'TRUE' }
VERSION : 0.1
// stored: InstanceOfName 03_FDBACK error
"03_FDBACK error"
BEGIN
END_DATA_BLOCK

DATA_BLOCK "FDBK_Error_n0085-uc29-el001-k30001_SN51_1"   // DB2087, F_DB
{ S7_Optimized_Access := 'TRUE' }
VERSION : 0.1
// stored: InstanceOfName 03_FDBACK error
"03_FDBACK error"
BEGIN
END_DATA_BLOCK

DATA_BLOCK "FDBK_Error_n0091-zp001-el001-k30001_SN51_1"   // DB2088, F_DB
{ S7_Optimized_Access := 'TRUE' }
VERSION : 0.1
// stored: InstanceOfName 03_FDBACK error
"03_FDBACK error"
BEGIN
END_DATA_BLOCK

DATA_BLOCK "FDBK_Error_n0091-zp001-el001-k30001_SN51_2"   // DB2089, F_DB
{ S7_Optimized_Access := 'TRUE' }
VERSION : 0.1
// stored: InstanceOfName 03_FDBACK error
"03_FDBACK error"
BEGIN
END_DATA_BLOCK

DATA_BLOCK "FDBK_Error_n0093-ug7-el001-k30001_SN51_1"   // DB2090, F_DB
{ S7_Optimized_Access := 'TRUE' }
VERSION : 0.1
// stored: InstanceOfName 03_FDBACK error
"03_FDBACK error"
BEGIN
END_DATA_BLOCK

DATA_BLOCK "FDBK_Error_n0093-ug7-el001-k30001_SN51_2"   // DB2091, F_DB
{ S7_Optimized_Access := 'TRUE' }
VERSION : 0.1
// stored: InstanceOfName 03_FDBACK error
"03_FDBACK error"
BEGIN
END_DATA_BLOCK

DATA_BLOCK "FDBK_Error_n0093-ug7-el001-k30001_SN51_3"   // DB2092, F_DB
{ S7_Optimized_Access := 'TRUE' }
VERSION : 0.1
// stored: InstanceOfName 03_FDBACK error
"03_FDBACK error"
BEGIN
END_DATA_BLOCK

// folder: 02_Speed Control

DATA_BLOCK "Speed_Control_DB"   // DB17, F_DB
{ S7_Optimized_Access := 'TRUE' }
VERSION : 0.1
// stored: InstanceOfName 01_Speed_Control
"01_Speed_Control"
BEGIN
END_DATA_BLOCK

// folder: 03_Gate manager

DATA_BLOCK "MAINT_DOOR1"   // DB21, F_DB
{ S7_Optimized_Access := 'TRUE' }
VERSION : 0.1
// stored: InstanceOfName 02_Safety_Door
"02_Safety_Door"
BEGIN
END_DATA_BLOCK

// folder: (top level)

FUNCTION_BLOCK "Main_Safety_RTG1"   // FB1, F_FBD
{ S7_Optimized_Access := 'TRUE' }
   VAR_TEMP
      t_Reset : Bool;
   END_VAR
   VAR_TEMP   // added for the SCL form of the ladder/FBD networks
      _w1 : Bool;
      _w2 : Bool;
      _w3 : Bool;
      _w4 : Bool;
      _w5 : Bool;
      _w6 : Bool;
      _w7 : Bool;
      _w8 : Bool;
      _w9 : Bool;
   END_VAR
BEGIN

REGION Network 1: For commissioning
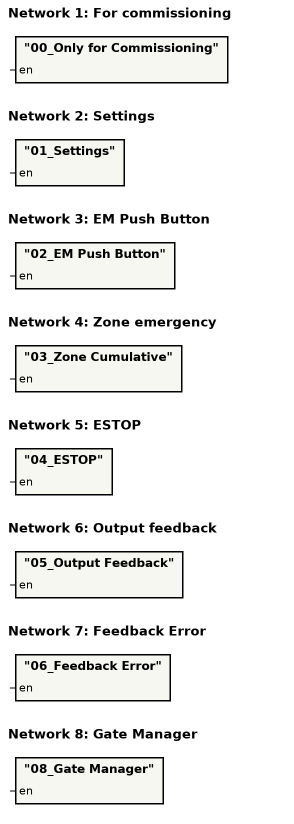
   "00_Only for Commissioning"();
END_REGION

REGION Network 2: Settings
   "01_Settings"();
END_REGION

REGION Network 3: EM Push Button
   "02_EM Push Button"();
END_REGION

REGION Network 4: Zone emergency
   "03_Zone Cumulative"();
END_REGION

REGION Network 5: ESTOP
   "04_ESTOP"();
END_REGION

REGION Network 6: Output feedback
   "05_Output Feedback"();
END_REGION

REGION Network 7: Feedback Error
   "06_Feedback Error"();
END_REGION

REGION Network 8: Gate Manager
   "08_Gate Manager"();
END_REGION

REGION Network 9: ACKNOWLEDGE ALARMS / RE-INTEGRATE FAULTY DEVICES OR PROGRAM BLOCKS
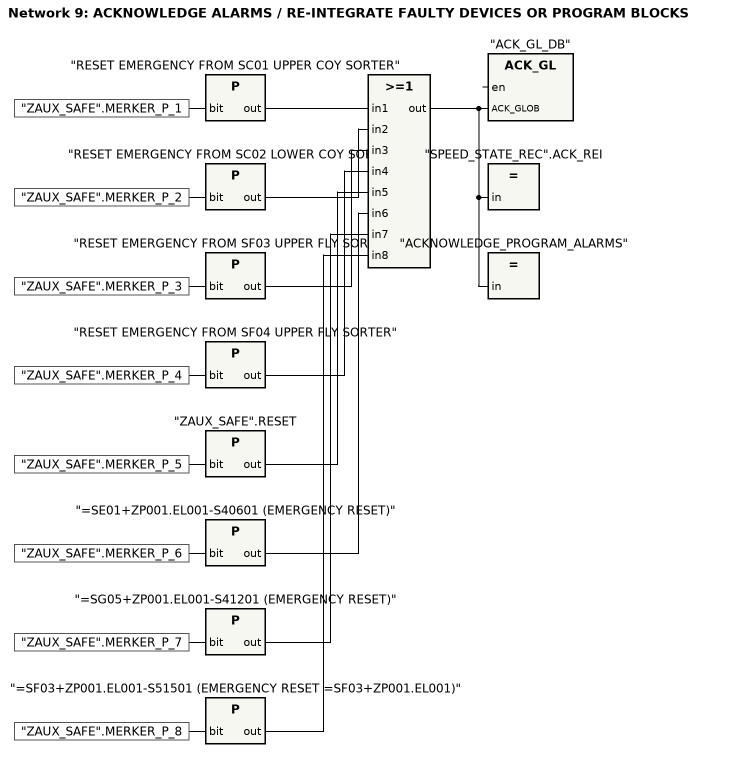
   #_w1 := "RESET EMERGENCY FROM SC01 UPPER COY SORTER" AND NOT "ZAUX_SAFE".MERKER_P_1;   // rising edge of "RESET EMERGENCY FROM SC01 UPPER COY SORTER"
   "ZAUX_SAFE".MERKER_P_1 := "RESET EMERGENCY FROM SC01 UPPER COY SORTER";
   #_w2 := "RESET EMERGENCY FROM SC02 LOWER COY SORTER" AND NOT "ZAUX_SAFE".MERKER_P_2;   // rising edge of "RESET EMERGENCY FROM SC02 LOWER COY SORTER"
   "ZAUX_SAFE".MERKER_P_2 := "RESET EMERGENCY FROM SC02 LOWER COY SORTER";
   #_w3 := "RESET EMERGENCY FROM SF03 UPPER FLY SORTER" AND NOT "ZAUX_SAFE".MERKER_P_3;   // rising edge of "RESET EMERGENCY FROM SF03 UPPER FLY SORTER"
   "ZAUX_SAFE".MERKER_P_3 := "RESET EMERGENCY FROM SF03 UPPER FLY SORTER";
   #_w4 := "RESET EMERGENCY FROM SF04 UPPER FLY SORTER" AND NOT "ZAUX_SAFE".MERKER_P_4;   // rising edge of "RESET EMERGENCY FROM SF04 UPPER FLY SORTER"
   "ZAUX_SAFE".MERKER_P_4 := "RESET EMERGENCY FROM SF04 UPPER FLY SORTER";
   #_w5 := "ZAUX_SAFE".RESET AND NOT "ZAUX_SAFE".MERKER_P_5;   // rising edge of "ZAUX_SAFE".RESET
   "ZAUX_SAFE".MERKER_P_5 := "ZAUX_SAFE".RESET;
   #_w6 := "=SE01+ZP001.EL001-S40601 (EMERGENCY RESET)" AND NOT "ZAUX_SAFE".MERKER_P_6;   // rising edge of "=SE01+ZP001.EL001-S40601 (EMERGENCY RESET)"
   "ZAUX_SAFE".MERKER_P_6 := "=SE01+ZP001.EL001-S40601 (EMERGENCY RESET)";
   #_w7 := "=SG05+ZP001.EL001-S41201 (EMERGENCY RESET)" AND NOT "ZAUX_SAFE".MERKER_P_7;   // rising edge of "=SG05+ZP001.EL001-S41201 (EMERGENCY RESET)"
   "ZAUX_SAFE".MERKER_P_7 := "=SG05+ZP001.EL001-S41201 (EMERGENCY RESET)";
   #_w8 := "=SF03+ZP001.EL001-S51501 (EMERGENCY RESET =SF03+ZP001.EL001)" AND NOT "ZAUX_SAFE".MERKER_P_8;   // rising edge of "=SF03+ZP001.EL001-S51501 (EMERGENCY RESET =SF03+ZP001.EL001)"
   "ZAUX_SAFE".MERKER_P_8 := "=SF03+ZP001.EL001-S51501 (EMERGENCY RESET =SF03+ZP001.EL001)";
   "SPEED_STATE_REC".ACK_REI := #_w1 OR #_w2 OR #_w3 OR #_w4 OR #_w5 OR #_w6 OR #_w7 OR #_w8;
   "ACKNOWLEDGE_PROGRAM_ALARMS" := "SPEED_STATE_REC".ACK_REI;
   "ACK_GL_DB"(ACK_GLOB := "SPEED_STATE_REC".ACK_REI);   // ACK_GL
END_REGION

REGION Network 10: RESET GLOBAL
   // Add any other reset
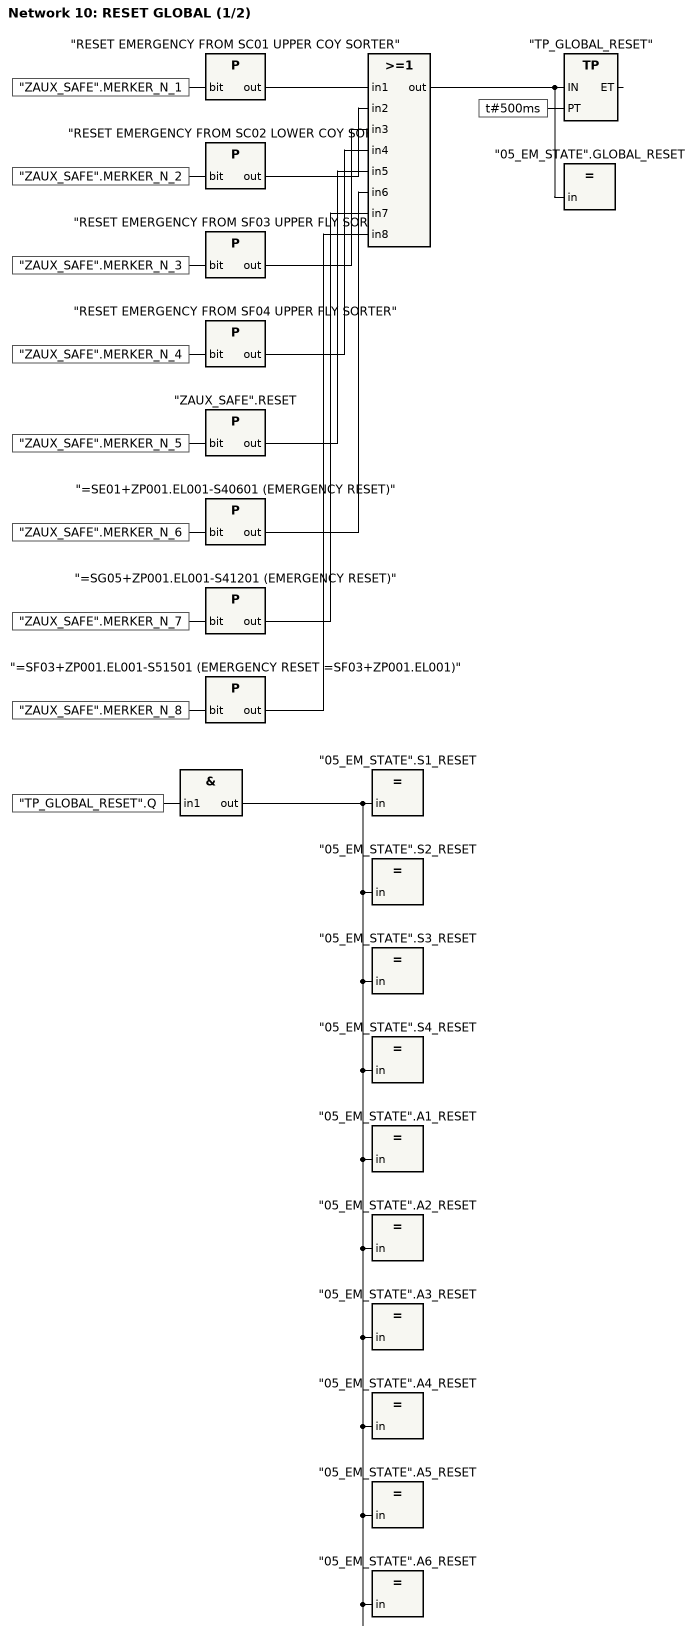
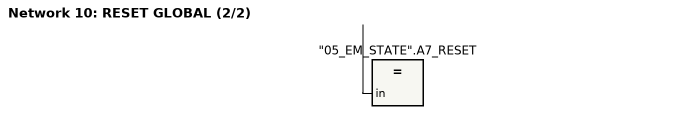
   #_w1 := "RESET EMERGENCY FROM SC01 UPPER COY SORTER" AND NOT "ZAUX_SAFE".MERKER_N_1;   // rising edge of "RESET EMERGENCY FROM SC01 UPPER COY SORTER"
   "ZAUX_SAFE".MERKER_N_1 := "RESET EMERGENCY FROM SC01 UPPER COY SORTER";
   #_w2 := "RESET EMERGENCY FROM SC02 LOWER COY SORTER" AND NOT "ZAUX_SAFE".MERKER_N_2;   // rising edge of "RESET EMERGENCY FROM SC02 LOWER COY SORTER"
   "ZAUX_SAFE".MERKER_N_2 := "RESET EMERGENCY FROM SC02 LOWER COY SORTER";
   #_w3 := "RESET EMERGENCY FROM SF03 UPPER FLY SORTER" AND NOT "ZAUX_SAFE".MERKER_N_3;   // rising edge of "RESET EMERGENCY FROM SF03 UPPER FLY SORTER"
   "ZAUX_SAFE".MERKER_N_3 := "RESET EMERGENCY FROM SF03 UPPER FLY SORTER";
   #_w4 := "RESET EMERGENCY FROM SF04 UPPER FLY SORTER" AND NOT "ZAUX_SAFE".MERKER_N_4;   // rising edge of "RESET EMERGENCY FROM SF04 UPPER FLY SORTER"
   "ZAUX_SAFE".MERKER_N_4 := "RESET EMERGENCY FROM SF04 UPPER FLY SORTER";
   #_w5 := "ZAUX_SAFE".RESET AND NOT "ZAUX_SAFE".MERKER_N_5;   // rising edge of "ZAUX_SAFE".RESET
   "ZAUX_SAFE".MERKER_N_5 := "ZAUX_SAFE".RESET;
   #_w6 := "=SE01+ZP001.EL001-S40601 (EMERGENCY RESET)" AND NOT "ZAUX_SAFE".MERKER_N_6;   // rising edge of "=SE01+ZP001.EL001-S40601 (EMERGENCY RESET)"
   "ZAUX_SAFE".MERKER_N_6 := "=SE01+ZP001.EL001-S40601 (EMERGENCY RESET)";
   #_w7 := "=SG05+ZP001.EL001-S41201 (EMERGENCY RESET)" AND NOT "ZAUX_SAFE".MERKER_N_7;   // rising edge of "=SG05+ZP001.EL001-S41201 (EMERGENCY RESET)"
   "ZAUX_SAFE".MERKER_N_7 := "=SG05+ZP001.EL001-S41201 (EMERGENCY RESET)";
   #_w8 := "=SF03+ZP001.EL001-S51501 (EMERGENCY RESET =SF03+ZP001.EL001)" AND NOT "ZAUX_SAFE".MERKER_N_8;   // rising edge of "=SF03+ZP001.EL001-S51501 (EMERGENCY RESET =SF03+ZP001.EL001)"
   "ZAUX_SAFE".MERKER_N_8 := "=SF03+ZP001.EL001-S51501 (EMERGENCY RESET =SF03+ZP001.EL001)";
   #_w9 := #_w1 OR #_w2 OR #_w3 OR #_w4 OR #_w5 OR #_w6 OR #_w7 OR #_w8;
   "TP_GLOBAL_RESET".TP(IN := #_w9, PT := t#500ms);
   "05_EM_STATE".GLOBAL_RESET := #_w9;
   "05_EM_STATE".S1_RESET := "TP_GLOBAL_RESET".Q;
   "05_EM_STATE".S2_RESET := "TP_GLOBAL_RESET".Q;
   "05_EM_STATE".S3_RESET := "TP_GLOBAL_RESET".Q;
   "05_EM_STATE".S4_RESET := "TP_GLOBAL_RESET".Q;
   "05_EM_STATE".A1_RESET := "TP_GLOBAL_RESET".Q;
   "05_EM_STATE".A2_RESET := "TP_GLOBAL_RESET".Q;
   "05_EM_STATE".A3_RESET := "TP_GLOBAL_RESET".Q;
   "05_EM_STATE".A4_RESET := "TP_GLOBAL_RESET".Q;
   "05_EM_STATE".A5_RESET := "TP_GLOBAL_RESET".Q;
   "05_EM_STATE".A6_RESET := "TP_GLOBAL_RESET".Q;
   "05_EM_STATE".A7_RESET := "TP_GLOBAL_RESET".Q;
END_REGION

REGION Network 11: RESET LOCAL
END_REGION
END_FUNCTION_BLOCK

FUNCTION_BLOCK "00_Push-Button_Input"   // FB2, F_LAD
TITLE = Push-Button_Input_ET200
{ S7_Optimized_Access := 'TRUE' }
VERSION : 0.1
// Input
// Bypass_ET200
// IN_1
// IN_2
// IN_3
// IN_4
// ON_Diag
// ON_Lamp
// Reset
// Output
// OUT_1
// OUT_2
// OUT_3
// OUT_4
// Diag_1
// Diag_2
// Diag_3
// Diag_4
// Lamp_1
// Lamp_2
// Lamp_3
// Lamp_4
// 
// InOut
// 
// Static
// ESTOP_1
// ESTOP_2
// ESTOP_3
// ESTOP_4
// Temp
// 
// Constant
   VAR_INPUT
      IN_1 : Bool;
      IN_2 : Bool;
      IN_3 : Bool;
      IN_4 : Bool;
      ON_Tristate : Bool;
      ON_Lamp : Bool;
      Reset : Bool;
      REAC_DELAY : Time := T#500ms;   // Reactivation delay= the OUT goes from 0 to 1 after this time
      Bypass_ET200 : Bool;
   END_VAR
   VAR_OUTPUT
      OUT_1 : Bool;
      OUT_2 : Bool;
      OUT_3 : Bool;
      OUT_4 : Bool;
      Diag_1 : Bool;
      Diag_2 : Bool;
      Diag_3 : Bool;
      Diag_4 : Bool;
      Lamp_1 : Bool;
      Lamp_2 : Bool;
      Lamp_3 : Bool;
      Lamp_4 : Bool;
   END_VAR
   VAR
      ESTOP_1 : ESTOP1;
      ESTOP_2 : ESTOP1;
      ESTOP_3 : ESTOP1;
      ESTOP_4 : ESTOP1;
      TON_1 : TON;
      TON_2 : TON;
      TON_3 : TON;
      TON_4 : TON;
   END_VAR
BEGIN

REGION Network 1 (F_FBD): Card: 4 Input safety for Push-Button
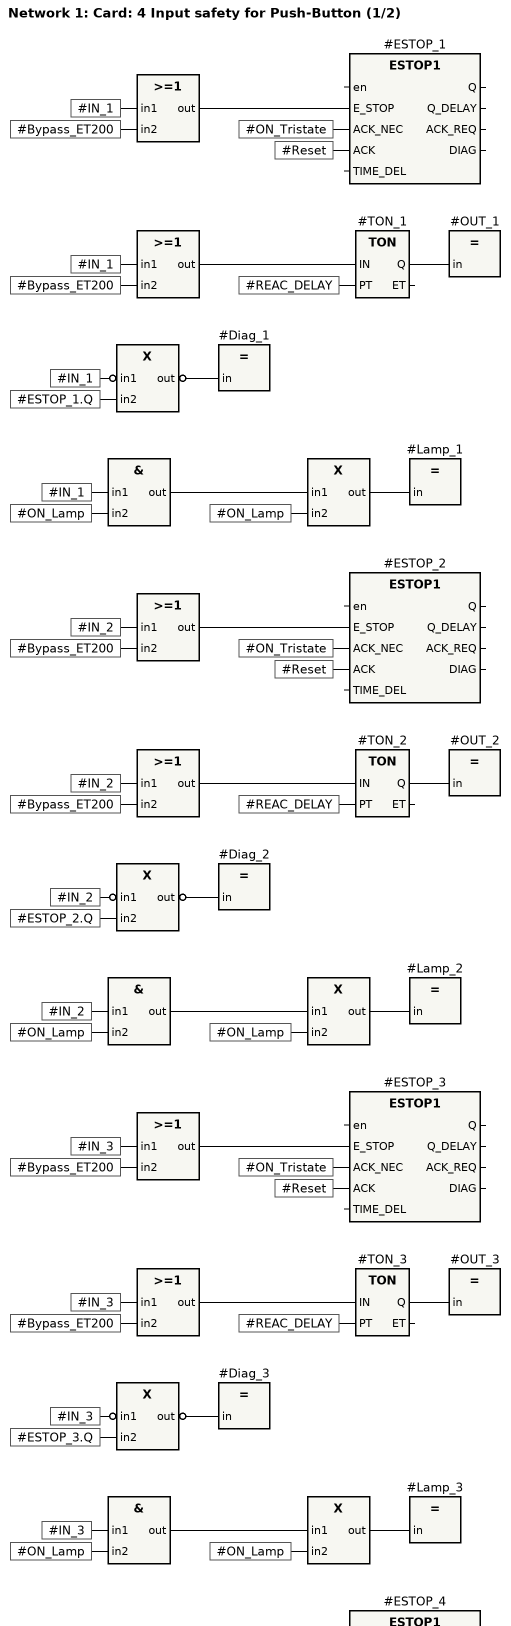
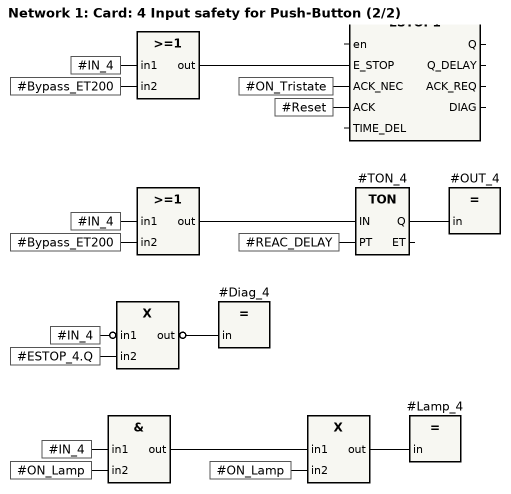
   #ESTOP_1(E_STOP := #IN_1 OR #Bypass_ET200, ACK_NEC := #ON_Tristate, ACK := #Reset);   // ESTOP1
   #TON_1.TON(IN := #IN_1 OR #Bypass_ET200, PT := #REAC_DELAY);
   #OUT_1 := #TON_1.Q;
   #Diag_1 := NOT (NOT #IN_1 XOR #ESTOP_1.Q);
   #Lamp_1 := (#IN_1 AND #ON_Lamp) XOR #ON_Lamp;
   #ESTOP_2(E_STOP := #IN_2 OR #Bypass_ET200, ACK_NEC := #ON_Tristate, ACK := #Reset);   // ESTOP1
   #TON_2.TON(IN := #IN_2 OR #Bypass_ET200, PT := #REAC_DELAY);
   #OUT_2 := #TON_2.Q;
   #Diag_2 := NOT (NOT #IN_2 XOR #ESTOP_2.Q);
   #Lamp_2 := (#IN_2 AND #ON_Lamp) XOR #ON_Lamp;
   #ESTOP_3(E_STOP := #IN_3 OR #Bypass_ET200, ACK_NEC := #ON_Tristate, ACK := #Reset);   // ESTOP1
   #TON_3.TON(IN := #IN_3 OR #Bypass_ET200, PT := #REAC_DELAY);
   #OUT_3 := #TON_3.Q;
   #Diag_3 := NOT (NOT #IN_3 XOR #ESTOP_3.Q);
   #Lamp_3 := (#IN_3 AND #ON_Lamp) XOR #ON_Lamp;
   #ESTOP_4(E_STOP := #IN_4 OR #Bypass_ET200, ACK_NEC := #ON_Tristate, ACK := #Reset);   // ESTOP1
   #TON_4.TON(IN := #IN_4 OR #Bypass_ET200, PT := #REAC_DELAY);
   #OUT_4 := #TON_4.Q;
   #Diag_4 := NOT (NOT #IN_4 XOR #ESTOP_4.Q);
   #Lamp_4 := (#IN_4 AND #ON_Lamp) XOR #ON_Lamp;
END_REGION
END_FUNCTION_BLOCK

FUNCTION_BLOCK "01_Speed_Control"   // FB3, F_FBD
{ S7_Optimized_Access := 'TRUE' }
VERSION : 0.1
   VAR_INPUT
      "Sorter in RUN" : Bool;   // Sorter in Run from sorter
      PH1 : Bool;   // Phisycal input PH1
      PH2 : Bool;   // Phisycal input PH2
      "Time" : Time := T#4s;   // Time used to check the state of the sorter
      Running_Delay : Time := T#5s;   // Delay to sorter running
   END_VAR
   VAR_OUTPUT
      "Sorter STOP" : Bool;
      "Broken PH safety encoder" : Bool;
      "Stop PH1" : Bool;
      "Stop PH2" : Bool;
      "Broken PH1" : Bool;
      "Broken PH2" : Bool;
   END_VAR
   VAR
      TON_Stop1_PH1 : TON;
      TON_Stop2_PH1 : TON;
      TON_Broken1_PH1 : TON;
      TON_Broken2_PH1 : TON;
      TON_Stop1_PH2 : TON;
      TON_Stop2_PH2 : TON;
      TON_Broken1_PH2 : TON;
      TON_Broken2_PH2 : TON;
      TON_SORTER_DELAY : TON;
   END_VAR
   VAR_TEMP
      "t_Stop PH1_temp" : Bool;
      "t_Stop PH2_temp" : Bool;
      "t_Broken PH1_temp" : Bool;
      "t_Broken PH2_temp" : Bool;
      t_Sorter_Running : Bool;
   END_VAR
   VAR_TEMP   // added for the SCL form of the ladder/FBD networks
      _w1 : Bool;
   END_VAR
BEGIN

REGION Network 1
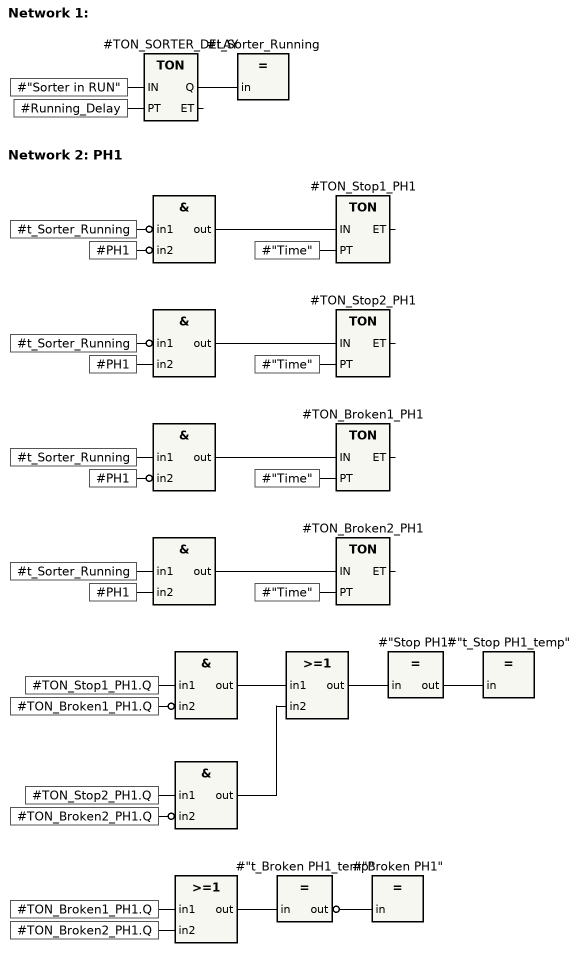
   #TON_SORTER_DELAY.TON(IN := #"Sorter in RUN", PT := #Running_Delay);
   #t_Sorter_Running := #TON_SORTER_DELAY.Q;
END_REGION

REGION Network 2: PH1
   #TON_Stop1_PH1.TON(IN := NOT #t_Sorter_Running AND NOT #PH1, PT := #"Time");
   #TON_Stop2_PH1.TON(IN := NOT #t_Sorter_Running AND #PH1, PT := #"Time");
   #TON_Broken1_PH1.TON(IN := #t_Sorter_Running AND NOT #PH1, PT := #"Time");
   #TON_Broken2_PH1.TON(IN := #t_Sorter_Running AND #PH1, PT := #"Time");
   #"Stop PH1" := (#TON_Stop1_PH1.Q AND NOT #TON_Broken1_PH1.Q) OR (#TON_Stop2_PH1.Q AND NOT #TON_Broken2_PH1.Q);
   #"t_Stop PH1_temp" := #"Stop PH1";
   #_w1 := #TON_Broken1_PH1.Q OR #TON_Broken2_PH1.Q;
   #"t_Broken PH1_temp" := #_w1;
   #"Broken PH1" := NOT #_w1;
END_REGION

REGION Network 3: PH2
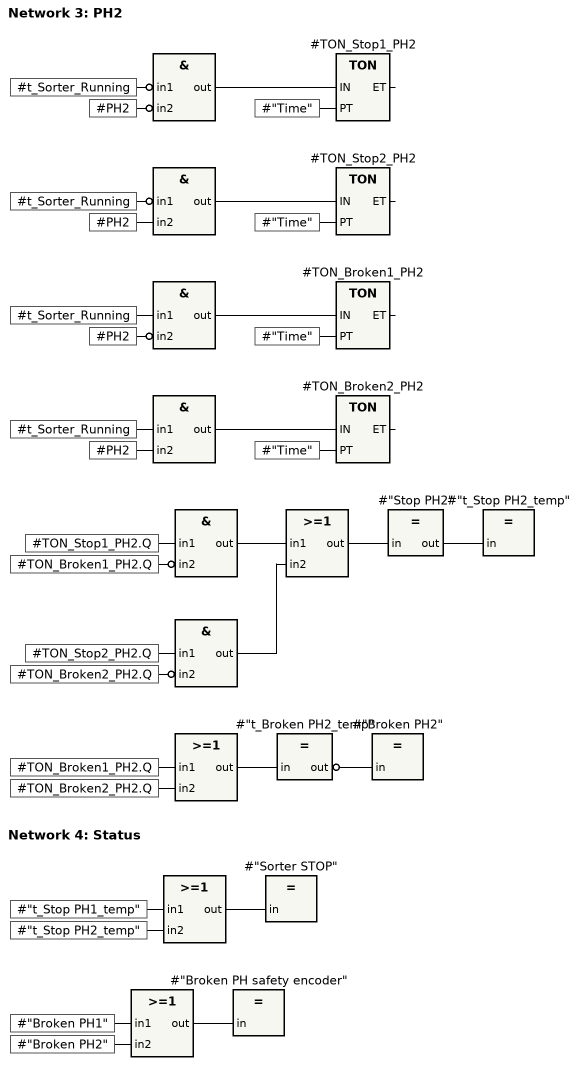
   #TON_Stop1_PH2.TON(IN := NOT #t_Sorter_Running AND NOT #PH2, PT := #"Time");
   #TON_Stop2_PH2.TON(IN := NOT #t_Sorter_Running AND #PH2, PT := #"Time");
   #TON_Broken1_PH2.TON(IN := #t_Sorter_Running AND NOT #PH2, PT := #"Time");
   #TON_Broken2_PH2.TON(IN := #t_Sorter_Running AND #PH2, PT := #"Time");
   #"Stop PH2" := (#TON_Stop1_PH2.Q AND NOT #TON_Broken1_PH2.Q) OR (#TON_Stop2_PH2.Q AND NOT #TON_Broken2_PH2.Q);
   #"t_Stop PH2_temp" := #"Stop PH2";
   #_w1 := #TON_Broken1_PH2.Q OR #TON_Broken2_PH2.Q;
   #"t_Broken PH2_temp" := #_w1;
   #"Broken PH2" := NOT #_w1;
END_REGION

REGION Network 4: Status
   #"Sorter STOP" := #"t_Stop PH1_temp" OR #"t_Stop PH2_temp";
   #"Broken PH safety encoder" := #"Broken PH1" OR #"Broken PH2";
END_REGION
END_FUNCTION_BLOCK

FUNCTION_BLOCK "03_FDBACK error"   // FB4, F_LAD
TITLE = 03_FDBACK error
{ S7_Optimized_Access := 'TRUE' }
VERSION : 0.1
// Input
// Commissioning_bypass
// FDBACK ERROR 1
// FDBACK ERROR 2
// FDBACK ERROR 3
// FDBACK ERROR 4
// FDBACK ERROR 5
// FDBACK ERROR 6
// FDBACK ERROR 7
// FDBACK ERROR 8
// FDBACK ERROR 9
// FDBACK ERROR 10
// 
// Output
// Cumulative FDBACK
// 
// InOut
// 
// Static
// 
// Temp
// 
// Constant
   VAR_INPUT
      Commissioning_bypass : Bool;
      "FDBACK ERROR 1" : Bool;
      "FDBACK ERROR 2" : Bool;
      "FDBACK ERROR 3" : Bool;
      "FDBACK ERROR 4" : Bool;
      "FDBACK ERROR 5" : Bool;
      "FDBACK ERROR 6" : Bool;
      "FDBACK ERROR 7" : Bool;
      "FDBACK ERROR 8" : Bool;
   END_VAR
   VAR_OUTPUT
      "Cumulative FDBACK" : Bool;
      "ERROR 1" : Bool;
      "ERROR 2" : Bool;
      "ERROR 3" : Bool;
      "ERROR 4" : Bool;
      "ERROR 5" : Bool;
      "ERROR 6" : Bool;
      "ERROR 7" : Bool;
      "ERROR 8" : Bool;
   END_VAR
BEGIN

REGION Network 1: First channel
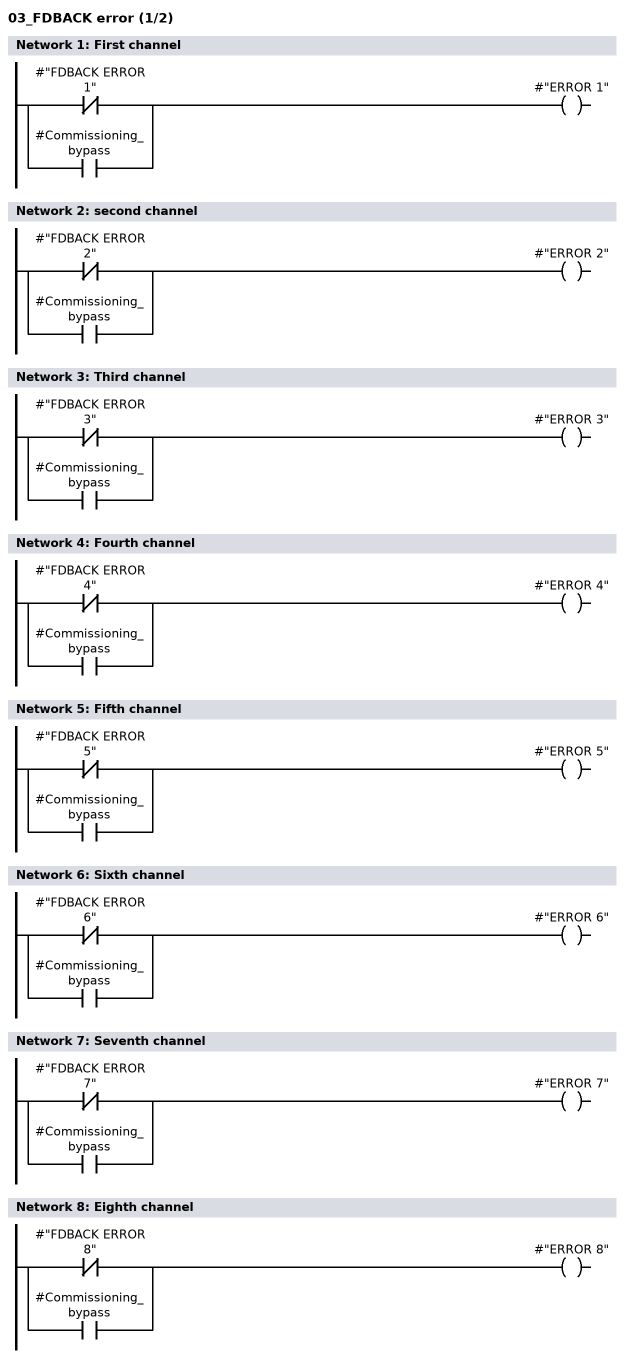
   RUNG wire#powerrail
      I_Contact( #"FDBACK ERROR 1" )
      wire#w1
      Coil( #"ERROR 1" )
   END_RUNG
   RUNG wire#powerrail
      Contact( #Commissioning_bypass )
   END_RUNG wire#w1
   // the same network as SCL:
   #"ERROR 1" := NOT #"FDBACK ERROR 1" OR #Commissioning_bypass;
END_REGION

REGION Network 2: second channel
   RUNG wire#powerrail
      I_Contact( #"FDBACK ERROR 2" )
      wire#w1
      Coil( #"ERROR 2" )
   END_RUNG
   RUNG wire#powerrail
      Contact( #Commissioning_bypass )
   END_RUNG wire#w1
   // the same network as SCL:
   #"ERROR 2" := NOT #"FDBACK ERROR 2" OR #Commissioning_bypass;
END_REGION

REGION Network 3: Third channel
   RUNG wire#powerrail
      I_Contact( #"FDBACK ERROR 3" )
      wire#w1
      Coil( #"ERROR 3" )
   END_RUNG
   RUNG wire#powerrail
      Contact( #Commissioning_bypass )
   END_RUNG wire#w1
   // the same network as SCL:
   #"ERROR 3" := NOT #"FDBACK ERROR 3" OR #Commissioning_bypass;
END_REGION

REGION Network 4: Fourth channel
   RUNG wire#powerrail
      I_Contact( #"FDBACK ERROR 4" )
      wire#w1
      Coil( #"ERROR 4" )
   END_RUNG
   RUNG wire#powerrail
      Contact( #Commissioning_bypass )
   END_RUNG wire#w1
   // the same network as SCL:
   #"ERROR 4" := NOT #"FDBACK ERROR 4" OR #Commissioning_bypass;
END_REGION

REGION Network 5: Fifth channel
   RUNG wire#powerrail
      I_Contact( #"FDBACK ERROR 5" )
      wire#w1
      Coil( #"ERROR 5" )
   END_RUNG
   RUNG wire#powerrail
      Contact( #Commissioning_bypass )
   END_RUNG wire#w1
   // the same network as SCL:
   #"ERROR 5" := NOT #"FDBACK ERROR 5" OR #Commissioning_bypass;
END_REGION

REGION Network 6: Sixth channel
   RUNG wire#powerrail
      I_Contact( #"FDBACK ERROR 6" )
      wire#w1
      Coil( #"ERROR 6" )
   END_RUNG
   RUNG wire#powerrail
      Contact( #Commissioning_bypass )
   END_RUNG wire#w1
   // the same network as SCL:
   #"ERROR 6" := NOT #"FDBACK ERROR 6" OR #Commissioning_bypass;
END_REGION

REGION Network 7: Seventh channel
   RUNG wire#powerrail
      I_Contact( #"FDBACK ERROR 7" )
      wire#w1
      Coil( #"ERROR 7" )
   END_RUNG
   RUNG wire#powerrail
      Contact( #Commissioning_bypass )
   END_RUNG wire#w1
   // the same network as SCL:
   #"ERROR 7" := NOT #"FDBACK ERROR 7" OR #Commissioning_bypass;
END_REGION

REGION Network 8: Eighth channel
   RUNG wire#powerrail
      I_Contact( #"FDBACK ERROR 8" )
      wire#w1
      Coil( #"ERROR 8" )
   END_RUNG
   RUNG wire#powerrail
      Contact( #Commissioning_bypass )
   END_RUNG wire#w1
   // the same network as SCL:
   #"ERROR 8" := NOT #"FDBACK ERROR 8" OR #Commissioning_bypass;
END_REGION

REGION Network 9: Cumulative error
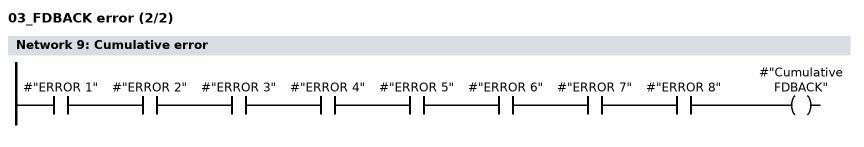
   RUNG wire#powerrail
      Contact( #"ERROR 1" )
      Contact( #"ERROR 2" )
      Contact( #"ERROR 3" )
      Contact( #"ERROR 4" )
      Contact( #"ERROR 5" )
      Contact( #"ERROR 6" )
      Contact( #"ERROR 7" )
      Contact( #"ERROR 8" )
      Coil( #"Cumulative FDBACK" )
   END_RUNG
   // the same network as SCL:
   #"Cumulative FDBACK" := #"ERROR 1" AND #"ERROR 2" AND #"ERROR 3" AND #"ERROR 4" AND #"ERROR 5" AND #"ERROR 6" AND #"ERROR 7" AND #"ERROR 8";
END_REGION
END_FUNCTION_BLOCK

FUNCTION_BLOCK "02_Safety_Door"   // FB5, F_LAD
{ S7_Optimized_Access := 'TRUE' }
VERSION : 0.1
   VAR_INPUT
      Bypass_For_Commissioning : Bool;
      DIAG : Bool := TRUE;
      CH1 : Bool := TRUE;
      CH2 : Bool := TRUE;
      "1oo1_evaluation" : Bool;   // Manage the 2 channels separately
      "Sorter_Running_from MSC" : Bool;
      Sorter_Stop_from_Encoder : Bool;
      Open_Request : Bool;
      Alarm_Filter : Bool;
      Sorter_Door : Bool := TRUE;
      ACK_NEC : Bool;   // For non sorter doors
      ACK : Bool;   // For non sorter doors
   END_VAR
   VAR_OUTPUT
      Solenoid : Bool;
      EM_Cut : Bool;
      EM_Cut_Delay : Bool;
      Diag_Open : Bool;
      Diag_Alarm : Bool;
   END_VAR
   VAR
      "E-STOP" : ESTOP1;
      TON_Alarm : TON;
   END_VAR
   VAR_TEMP
      Alarm_Temp : Bool;
      t_ALARM : Bool;
   END_VAR
BEGIN

REGION Network 1: Emergency cut
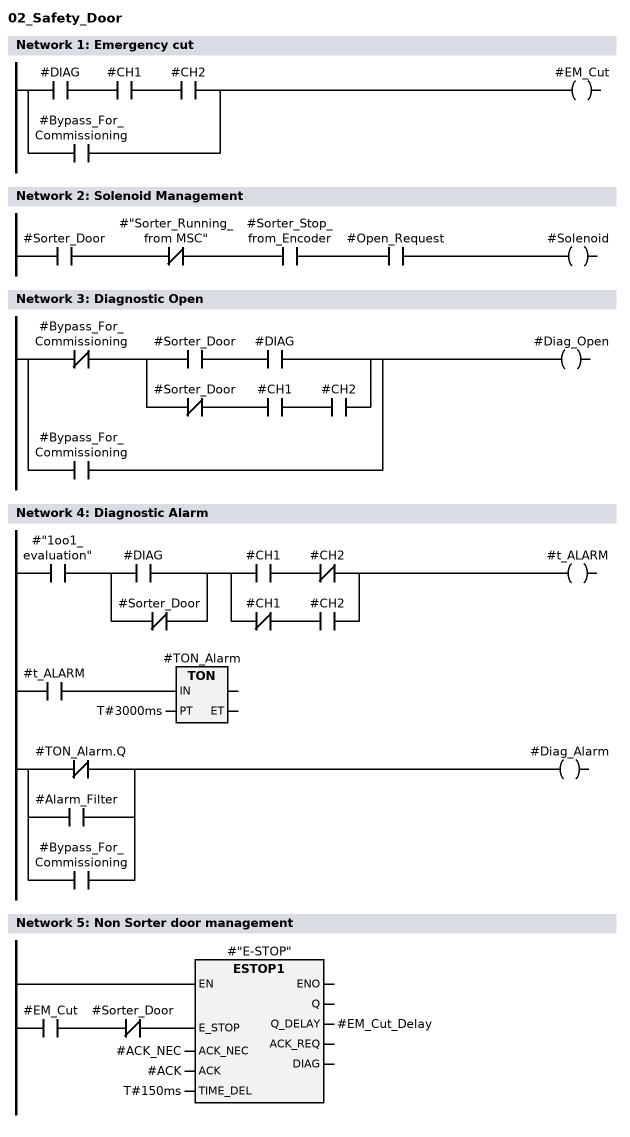
   RUNG wire#powerrail
      Contact( #DIAG )
      Contact( #CH1 )
      Contact( #CH2 )
      wire#w1
      Coil( #EM_Cut )
   END_RUNG
   RUNG wire#powerrail
      Contact( #Bypass_For_Commissioning )
   END_RUNG wire#w1
   // the same network as SCL:
   #EM_Cut := (#DIAG AND #CH1 AND #CH2) OR #Bypass_For_Commissioning;
END_REGION

REGION Network 2: Solenoid Management
   RUNG wire#powerrail
      Contact( #Sorter_Door )
      I_Contact( #"Sorter_Running_from MSC" )
      Contact( #Sorter_Stop_from_Encoder )
      Contact( #Open_Request )
      Coil( #Solenoid )
   END_RUNG
   // the same network as SCL:
   #Solenoid := #Sorter_Door AND NOT #"Sorter_Running_from MSC" AND #Sorter_Stop_from_Encoder AND #Open_Request;
END_REGION

REGION Network 3: Diagnostic Open
   RUNG wire#powerrail
      I_Contact( #Bypass_For_Commissioning )
      wire#w1
      Contact( #Sorter_Door )
      Contact( #DIAG )
      wire#w2
      Coil( #Diag_Open )
   END_RUNG
   RUNG wire#w1
      I_Contact( #Sorter_Door )
      Contact( #CH1 )
      Contact( #CH2 )
   END_RUNG wire#w2
   RUNG wire#powerrail
      Contact( #Bypass_For_Commissioning )
   END_RUNG wire#w2
   // the same network as SCL:
   #Diag_Open := (NOT #Bypass_For_Commissioning AND ((#Sorter_Door AND #DIAG) OR (NOT #Sorter_Door AND #CH1 AND #CH2))) OR #Bypass_For_Commissioning;
END_REGION

REGION Network 4: Diagnostic Alarm
   #t_ALARM := #"1oo1_evaluation" AND (#DIAG OR NOT #Sorter_Door) AND ((#CH1 AND NOT #CH2) OR (NOT #CH1 AND #CH2));
   #TON_Alarm.TON(IN := #t_ALARM, PT := T#3000ms);
   #Diag_Alarm := NOT #TON_Alarm.Q OR #Alarm_Filter OR #Bypass_For_Commissioning;
END_REGION

REGION Network 5: Non Sorter door management
   #"E-STOP"(E_STOP := #EM_Cut AND NOT #Sorter_Door,   // ESTOP1
             ACK_NEC := #ACK_NEC,
             ACK := #ACK,
             TIME_DEL := T#150ms,
             Q_DELAY => #EM_Cut_Delay);
END_REGION
END_FUNCTION_BLOCK

FUNCTION_BLOCK "01_Speed_Control_SLS"   // FB7, F_LAD
{ S7_Optimized_Access := 'TRUE' }
VERSION : 0.1
   VAR_INPUT
      PH1 : Bool;
      PH2 : Bool;
      SORTER_RUNNING_MSC : Bool;
      SLS_NOT_EN : Bool;
      "MIN[time]" : Time;   // SLS Limit[ms] = Blade length[mm] / Speed[mm/s]
      "MAX[time]" : Time := T#4s;   // Sorter not moving
      "DelayRunning[time]" : Time := T#5s;   // Delay running status from sorter
   END_VAR
   VAR_OUTPUT
      SPEED_ZERO : Bool;
      SPEED_TOOHIGH : Bool;
      "PH1 Broken" : Bool;
      "PH2 Broken" : Bool;
      ENC_BROKEN : Bool;
   END_VAR
   VAR_IN_OUT
      SLS_DATA : "SLS_DATA";
   END_VAR
   VAR
      Time_Limit : Time := T#10s;
      TON_SLS_T_PH1 : TON;
      TON_SLS_T_PH2 : TON;
      TOF_PH1_WORKING : TOF;
      TOF_PH2_WORKING : TOF;
      TON_SORTER_STOP : TON;
      TON_TIMEOUT_COUNT : TON;
      TON_DELAY_RUNNING_STATUS : TON;
      CTU_SLS_PH1 : CTU;
      CTU_SLS_PH2 : CTU;
   END_VAR
   VAR_TEMP
      t_SpeedTH_PH1 : Bool;
      t_SpeedTH_PH2 : Bool;
      t_Speed0_PH1 : Bool;
      t_Speed0_PH2 : Bool;
      t_PH1_FE : Bool;
      t_PH2_FE : Bool;
      t_PH1_RE : Bool;
      t_PH2_RE : Bool;
      t_PH1_BRK : Bool;
      t_PH2_BRK : Bool;
      t_SorterRunning : Bool;
   END_VAR
   VAR CONSTANT
      NUM_STH : Int := 3;   // Number of blades with speed too high in TIMEOUT_CTU time
      TIMEOUT_CTU : Time := T#5s;   // Deltatime to count number of blades too fast
   END_VAR
   VAR_TEMP   // added for the SCL form of the ladder/FBD networks
      _w1 : Bool;
      _w2 : Bool;
   END_VAR
BEGIN

REGION Network 1: Falling Edges
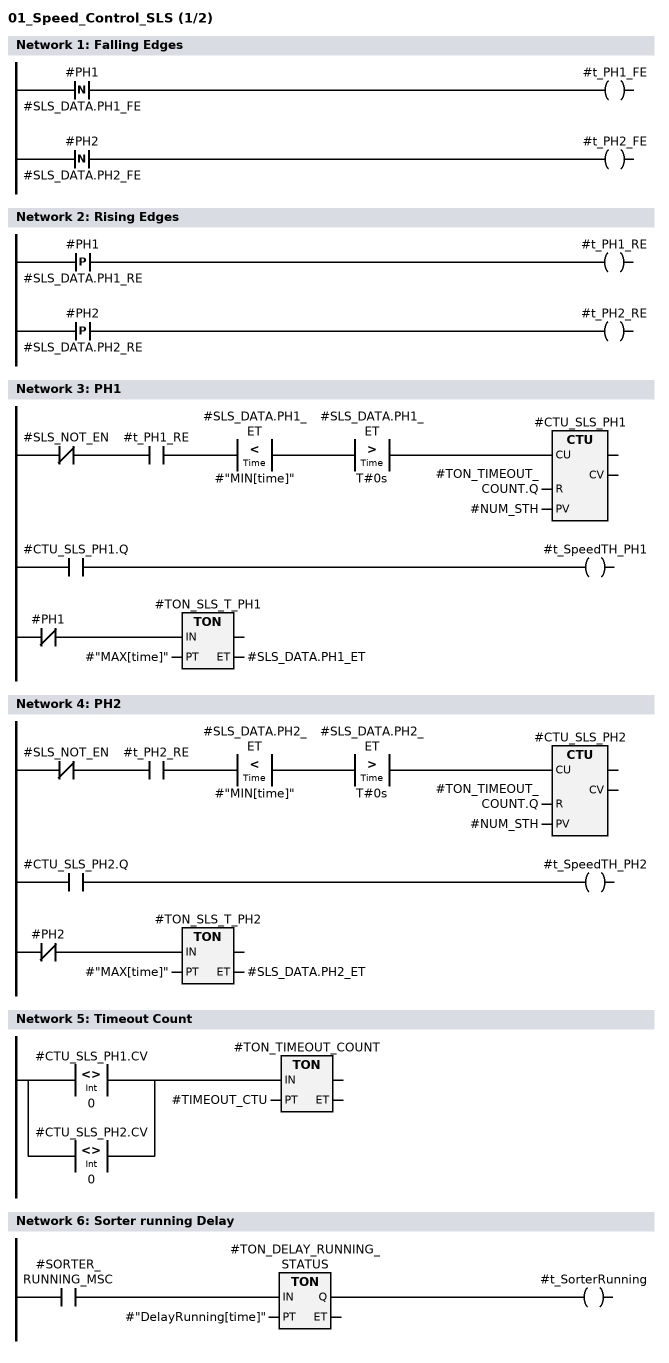
   RUNG wire#powerrail
      N_Contact(operand := #PH1, bit := #SLS_DATA.PH1_FE)
      Coil( #t_PH1_FE )
   END_RUNG
   RUNG wire#powerrail
      N_Contact(operand := #PH2, bit := #SLS_DATA.PH2_FE)
      Coil( #t_PH2_FE )
   END_RUNG
   // the same network as SCL:
   #_w1 := NOT #PH1 AND #SLS_DATA.PH1_FE;   // falling edge of #PH1
   #SLS_DATA.PH1_FE := #PH1;
   #t_PH1_FE := #_w1;
   #_w2 := NOT #PH2 AND #SLS_DATA.PH2_FE;   // falling edge of #PH2
   #SLS_DATA.PH2_FE := #PH2;
   #t_PH2_FE := #_w2;
END_REGION

REGION Network 2: Rising Edges
   RUNG wire#powerrail
      P_Contact(operand := #PH1, bit := #SLS_DATA.PH1_RE)
      Coil( #t_PH1_RE )
   END_RUNG
   RUNG wire#powerrail
      P_Contact(operand := #PH2, bit := #SLS_DATA.PH2_RE)
      Coil( #t_PH2_RE )
   END_RUNG
   // the same network as SCL:
   #_w1 := #PH1 AND NOT #SLS_DATA.PH1_RE;   // rising edge of #PH1
   #SLS_DATA.PH1_RE := #PH1;
   #t_PH1_RE := #_w1;
   #_w2 := #PH2 AND NOT #SLS_DATA.PH2_RE;   // rising edge of #PH2
   #SLS_DATA.PH2_RE := #PH2;
   #t_PH2_RE := #_w2;
END_REGION

REGION Network 3: PH1
   #CTU_SLS_PH1.CTU(CU := NOT #SLS_NOT_EN AND #t_PH1_RE AND (#SLS_DATA.PH1_ET < #"MIN[time]") AND (#SLS_DATA.PH1_ET > T#0s),
                    R := #TON_TIMEOUT_COUNT.Q,
                    PV := #NUM_STH);
   #t_SpeedTH_PH1 := #CTU_SLS_PH1.Q;
   #TON_SLS_T_PH1.TON(IN := NOT #PH1, PT := #"MAX[time]", ET => #SLS_DATA.PH1_ET);
END_REGION

REGION Network 4: PH2
   #CTU_SLS_PH2.CTU(CU := NOT #SLS_NOT_EN AND #t_PH2_RE AND (#SLS_DATA.PH2_ET < #"MIN[time]") AND (#SLS_DATA.PH2_ET > T#0s),
                    R := #TON_TIMEOUT_COUNT.Q,
                    PV := #NUM_STH);
   #t_SpeedTH_PH2 := #CTU_SLS_PH2.Q;
   #TON_SLS_T_PH2.TON(IN := NOT #PH2, PT := #"MAX[time]", ET => #SLS_DATA.PH2_ET);
END_REGION

REGION Network 5: Timeout Count
   #TON_TIMEOUT_COUNT.TON(IN := (#CTU_SLS_PH1.CV <> 0) OR (#CTU_SLS_PH2.CV <> 0), PT := #TIMEOUT_CTU);
END_REGION

REGION Network 6: Sorter running Delay
   #TON_DELAY_RUNNING_STATUS.TON(IN := #SORTER_RUNNING_MSC, PT := #"DelayRunning[time]");
   #t_SorterRunning := #TON_DELAY_RUNNING_STATUS.Q;
END_REGION

REGION Network 7: Speed too high
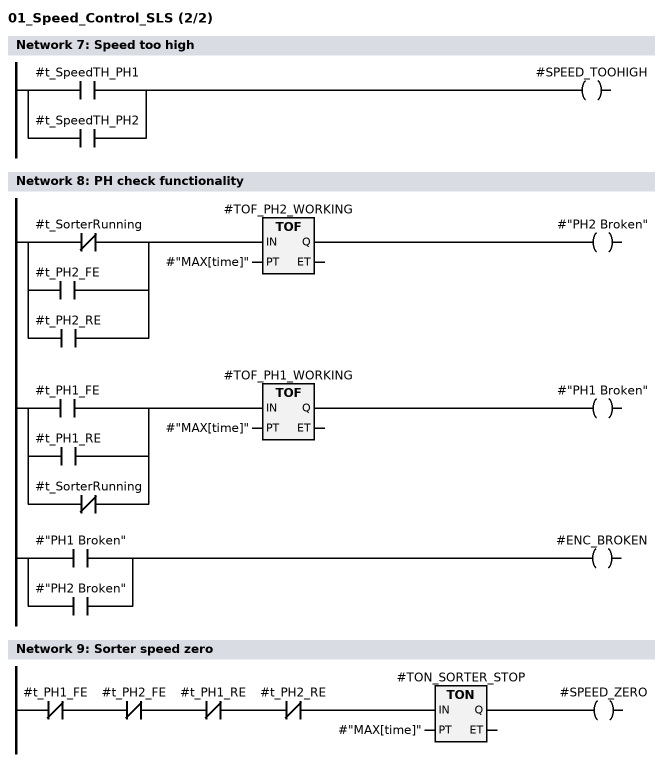
   RUNG wire#powerrail
      Contact( #t_SpeedTH_PH1 )
      wire#w1
      Coil( #SPEED_TOOHIGH )
   END_RUNG
   RUNG wire#powerrail
      Contact( #t_SpeedTH_PH2 )
   END_RUNG wire#w1
   // the same network as SCL:
   #SPEED_TOOHIGH := #t_SpeedTH_PH1 OR #t_SpeedTH_PH2;
END_REGION

REGION Network 8: PH check functionality
   #TOF_PH2_WORKING.TOF(IN := NOT #t_SorterRunning OR #t_PH2_FE OR #t_PH2_RE, PT := #"MAX[time]");
   #"PH2 Broken" := #TOF_PH2_WORKING.Q;
   #TOF_PH1_WORKING.TOF(IN := #t_PH1_FE OR #t_PH1_RE OR NOT #t_SorterRunning, PT := #"MAX[time]");
   #"PH1 Broken" := #TOF_PH1_WORKING.Q;
   #ENC_BROKEN := #"PH1 Broken" OR #"PH2 Broken";
END_REGION

REGION Network 9: Sorter speed zero
   #TON_SORTER_STOP.TON(IN := NOT #t_PH1_FE AND NOT #t_PH2_FE AND NOT #t_PH1_RE AND NOT #t_PH2_RE,
                        PT := #"MAX[time]");
   #SPEED_ZERO := #TON_SORTER_STOP.Q;
END_REGION
END_FUNCTION_BLOCK

FUNCTION_BLOCK "02_Safety_Door_Double_Sorter"   // FB10, F_LAD
{ S7_Optimized_Access := 'TRUE' }
VERSION : 0.1
   VAR_INPUT
      Bypass_For_Commissioning : Bool;
      DIAG : Bool := TRUE;
      CH1 : Bool := TRUE;
      CH2 : Bool := TRUE;
      "1oo1_evaluation" : Bool;   // Manage the 2 channels separately
      "Sorter1_Running_from MSC" : Bool;
      Sorter1_Stop_from_Encoder : Bool;
      Sorter1_Access_Allowed : Bool;
      "Sorter2_Running_from MSC" : Bool;
      Sorter2_Stop_from_Encoder : Bool;
      Sorter2_Access_Allowed : Bool;
      PB_Access_Request : Bool;
      Alarm_Filter : Bool;
   END_VAR
   VAR_OUTPUT
      Solenoid : Bool;
      EM_Cut : Bool;
      EM_Cut_Delay : Bool;
      Diag_Open : Bool;
      Diag_Alarm : Bool;
      Request_Access_to_Sorters : Bool;
      Access_Enabled_Lamp : Bool;
   END_VAR
   VAR
      "E-STOP" : ESTOP1;
      TON_Timeout_Request : TON;
      TON_Timeout_Opening : TON;
      TON_Alarm : TON;
      TON_Blink : TON;
      AuxBlink : Bool;
      Blink : Bool;
      Access_Enabled_Sorter1 : Bool;
      Access_Enabled_Sorter2 : Bool;
      Merker_Open_CMD : Bool;
      Merker_Access_Request : Bool;
      Merker_Blink : Bool;
      TON_Blink_Q : Bool;
   END_VAR
   VAR_TEMP
      Alarm_Temp : Bool;
      t_ALARM : Bool;
      Open_CMD : Bool;
   END_VAR
   VAR_TEMP   // added for the SCL form of the ladder/FBD networks
      _w1 : Bool;
   END_VAR
BEGIN

REGION Network 1: Emergency cut
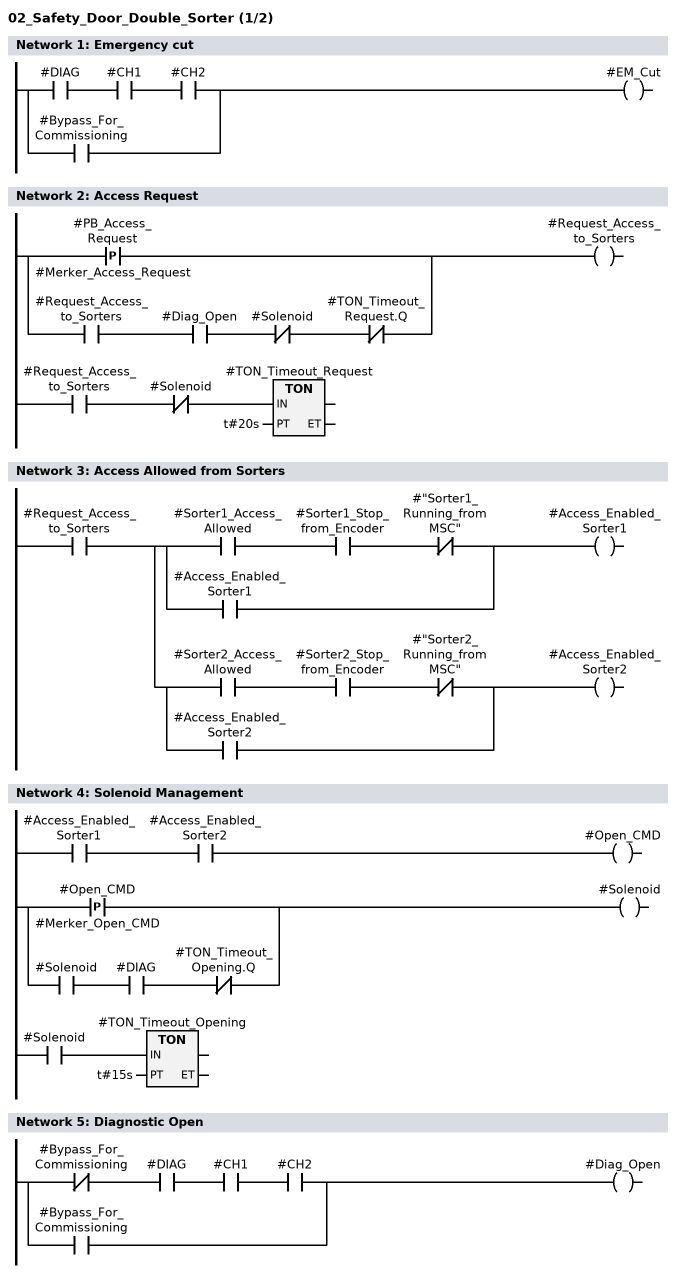
   RUNG wire#powerrail
      Contact( #DIAG )
      Contact( #CH1 )
      Contact( #CH2 )
      wire#w1
      Coil( #EM_Cut )
   END_RUNG
   RUNG wire#powerrail
      Contact( #Bypass_For_Commissioning )
   END_RUNG wire#w1
   // the same network as SCL:
   #EM_Cut := (#DIAG AND #CH1 AND #CH2) OR #Bypass_For_Commissioning;
END_REGION

REGION Network 2: Access Request
   #_w1 := #PB_Access_Request AND NOT #Merker_Access_Request;   // rising edge of #PB_Access_Request
   #Merker_Access_Request := #PB_Access_Request;
   #Request_Access_to_Sorters := #_w1 OR (#Request_Access_to_Sorters AND #Diag_Open AND NOT #Solenoid AND NOT #TON_Timeout_Request.Q);
   #TON_Timeout_Request.TON(IN := #Request_Access_to_Sorters AND NOT #Solenoid, PT := t#20s);
END_REGION

REGION Network 3: Access Allowed from Sorters
   RUNG wire#powerrail
      Contact( #Request_Access_to_Sorters )
      wire#w1
      Contact( #Sorter1_Access_Allowed )
      Contact( #Sorter1_Stop_from_Encoder )
      I_Contact( #"Sorter1_Running_from MSC" )
      wire#w2
      Coil( #Access_Enabled_Sorter1 )
   END_RUNG
   RUNG wire#w1
      Contact( #Access_Enabled_Sorter1 )
   END_RUNG wire#w2
   RUNG wire#w1
      Contact( #Sorter2_Access_Allowed )
      Contact( #Sorter2_Stop_from_Encoder )
      I_Contact( #"Sorter2_Running_from MSC" )
      wire#w3
      Coil( #Access_Enabled_Sorter2 )
   END_RUNG
   RUNG wire#w1
      Contact( #Access_Enabled_Sorter2 )
   END_RUNG wire#w3
   // the same network as SCL:
   #Access_Enabled_Sorter1 := #Request_Access_to_Sorters AND ((#Sorter1_Access_Allowed AND #Sorter1_Stop_from_Encoder AND NOT #"Sorter1_Running_from MSC") OR #Access_Enabled_Sorter1);
   #Access_Enabled_Sorter2 := #Request_Access_to_Sorters AND ((#Sorter2_Access_Allowed AND #Sorter2_Stop_from_Encoder AND NOT #"Sorter2_Running_from MSC") OR #Access_Enabled_Sorter2);
END_REGION

REGION Network 4: Solenoid Management
   #Open_CMD := #Access_Enabled_Sorter1 AND #Access_Enabled_Sorter2;
   #_w1 := #Open_CMD AND NOT #Merker_Open_CMD;   // rising edge of #Open_CMD
   #Merker_Open_CMD := #Open_CMD;
   #Solenoid := #_w1 OR (#Solenoid AND #DIAG AND NOT #TON_Timeout_Opening.Q);
   #TON_Timeout_Opening.TON(IN := #Solenoid, PT := t#15s);
END_REGION

REGION Network 5: Diagnostic Open
   RUNG wire#powerrail
      I_Contact( #Bypass_For_Commissioning )
      Contact( #DIAG )
      Contact( #CH1 )
      Contact( #CH2 )
      wire#w1
      Coil( #Diag_Open )
   END_RUNG
   RUNG wire#powerrail
      Contact( #Bypass_For_Commissioning )
   END_RUNG wire#w1
   // the same network as SCL:
   #Diag_Open := (NOT #Bypass_For_Commissioning AND #DIAG AND #CH1 AND #CH2) OR #Bypass_For_Commissioning;
END_REGION

REGION Network 6: Diagnostic Alarm
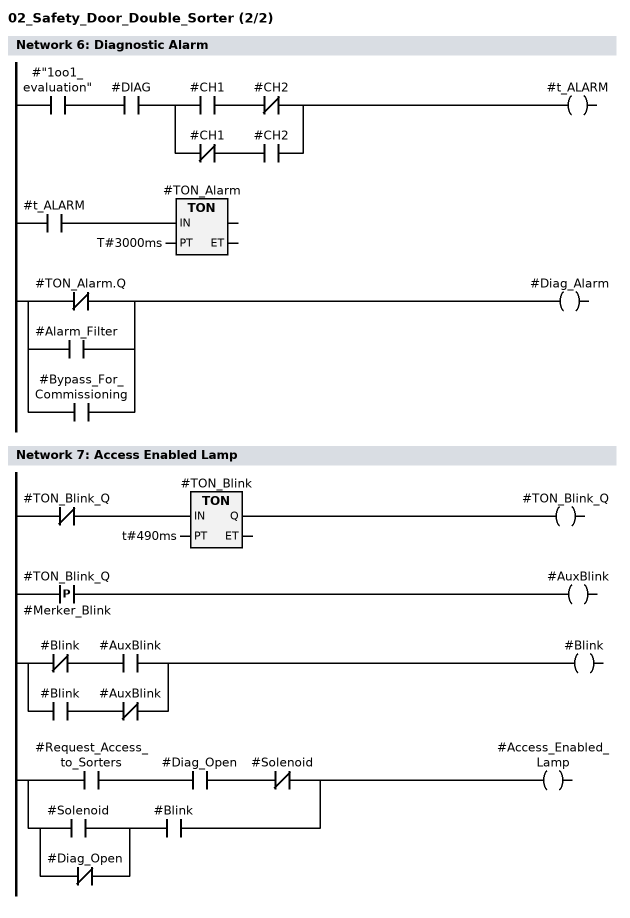
   #t_ALARM := #"1oo1_evaluation" AND #DIAG AND ((#CH1 AND NOT #CH2) OR (NOT #CH1 AND #CH2));
   #TON_Alarm.TON(IN := #t_ALARM, PT := T#3000ms);
   #Diag_Alarm := NOT #TON_Alarm.Q OR #Alarm_Filter OR #Bypass_For_Commissioning;
END_REGION

REGION Network 7: Access Enabled Lamp
   #TON_Blink.TON(IN := NOT #TON_Blink_Q, PT := t#490ms);
   #TON_Blink_Q := #TON_Blink.Q;
   #_w1 := #TON_Blink_Q AND NOT #Merker_Blink;   // rising edge of #TON_Blink_Q
   #Merker_Blink := #TON_Blink_Q;
   #AuxBlink := #_w1;
   #Blink := (NOT #Blink AND #AuxBlink) OR (#Blink AND NOT #AuxBlink);
   #Access_Enabled_Lamp := (#Request_Access_to_Sorters AND #Diag_Open AND NOT #Solenoid) OR ((#Solenoid OR NOT #Diag_Open) AND #Blink);
END_REGION
END_FUNCTION_BLOCK

FUNCTION "00_Only for Commissioning" : Void   // FC1, F_LAD
{ S7_Optimized_Access := 'TRUE' }
VERSION : 0.1
// Management of bypass to use during commissioning
BEGIN

REGION Network 1: Subnet50 Node0006
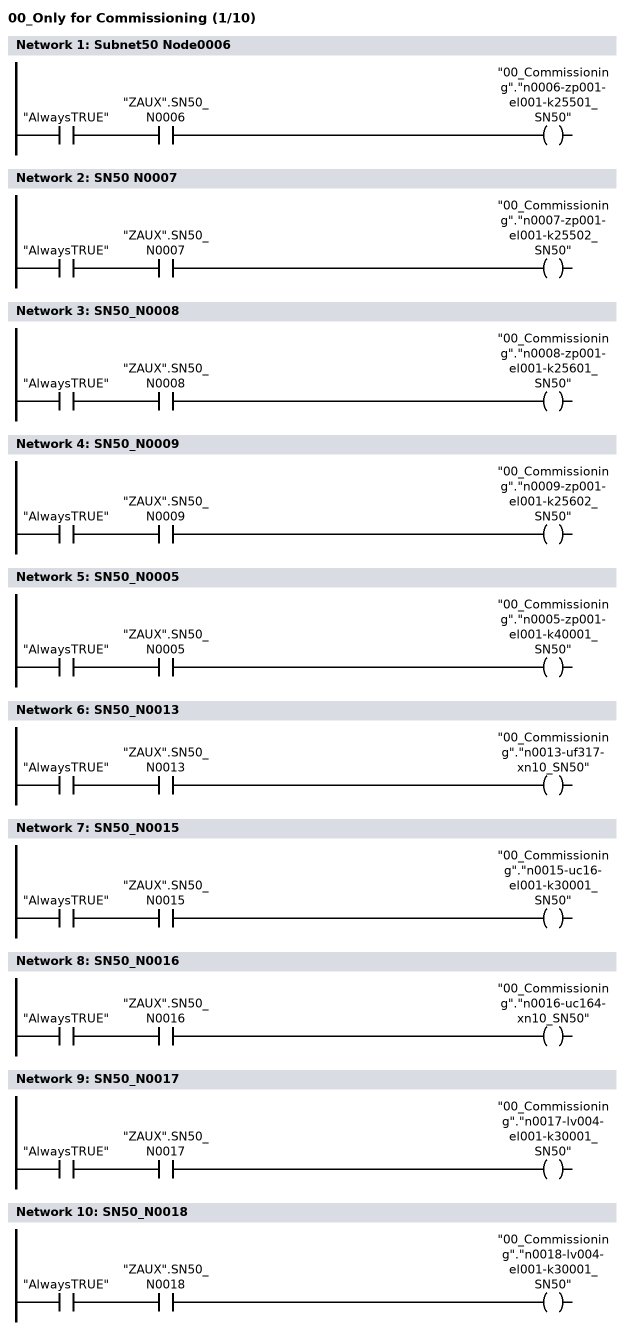
   RUNG wire#powerrail
      Contact( "AlwaysTRUE" )
      Contact( "ZAUX".SN50_N0006 )
      Coil( "00_Commissioning"."n0006-zp001-el001-k25501_SN50" )
   END_RUNG
   // the same network as SCL:
   "00_Commissioning"."n0006-zp001-el001-k25501_SN50" := "AlwaysTRUE" AND "ZAUX".SN50_N0006;
END_REGION

REGION Network 2: SN50 N0007
   RUNG wire#powerrail
      Contact( "AlwaysTRUE" )
      Contact( "ZAUX".SN50_N0007 )
      Coil( "00_Commissioning"."n0007-zp001-el001-k25502_SN50" )
   END_RUNG
   // the same network as SCL:
   "00_Commissioning"."n0007-zp001-el001-k25502_SN50" := "AlwaysTRUE" AND "ZAUX".SN50_N0007;
END_REGION

REGION Network 3: SN50_N0008
   RUNG wire#powerrail
      Contact( "AlwaysTRUE" )
      Contact( "ZAUX".SN50_N0008 )
      Coil( "00_Commissioning"."n0008-zp001-el001-k25601_SN50" )
   END_RUNG
   // the same network as SCL:
   "00_Commissioning"."n0008-zp001-el001-k25601_SN50" := "AlwaysTRUE" AND "ZAUX".SN50_N0008;
END_REGION

REGION Network 4: SN50_N0009
   RUNG wire#powerrail
      Contact( "AlwaysTRUE" )
      Contact( "ZAUX".SN50_N0009 )
      Coil( "00_Commissioning"."n0009-zp001-el001-k25602_SN50" )
   END_RUNG
   // the same network as SCL:
   "00_Commissioning"."n0009-zp001-el001-k25602_SN50" := "AlwaysTRUE" AND "ZAUX".SN50_N0009;
END_REGION

REGION Network 5: SN50_N0005
   RUNG wire#powerrail
      Contact( "AlwaysTRUE" )
      Contact( "ZAUX".SN50_N0005 )
      Coil( "00_Commissioning"."n0005-zp001-el001-k40001_SN50" )
   END_RUNG
   // the same network as SCL:
   "00_Commissioning"."n0005-zp001-el001-k40001_SN50" := "AlwaysTRUE" AND "ZAUX".SN50_N0005;
END_REGION

REGION Network 6: SN50_N0013
   RUNG wire#powerrail
      Contact( "AlwaysTRUE" )
      Contact( "ZAUX".SN50_N0013 )
      Coil( "00_Commissioning"."n0013-uf317-xn10_SN50" )
   END_RUNG
   // the same network as SCL:
   "00_Commissioning"."n0013-uf317-xn10_SN50" := "AlwaysTRUE" AND "ZAUX".SN50_N0013;
END_REGION

REGION Network 7: SN50_N0015
   RUNG wire#powerrail
      Contact( "AlwaysTRUE" )
      Contact( "ZAUX".SN50_N0015 )
      Coil( "00_Commissioning"."n0015-uc16-el001-k30001_SN50" )
   END_RUNG
   // the same network as SCL:
   "00_Commissioning"."n0015-uc16-el001-k30001_SN50" := "AlwaysTRUE" AND "ZAUX".SN50_N0015;
END_REGION

REGION Network 8: SN50_N0016
   RUNG wire#powerrail
      Contact( "AlwaysTRUE" )
      Contact( "ZAUX".SN50_N0016 )
      Coil( "00_Commissioning"."n0016-uc164-xn10_SN50" )
   END_RUNG
   // the same network as SCL:
   "00_Commissioning"."n0016-uc164-xn10_SN50" := "AlwaysTRUE" AND "ZAUX".SN50_N0016;
END_REGION

REGION Network 9: SN50_N0017
   RUNG wire#powerrail
      Contact( "AlwaysTRUE" )
      Contact( "ZAUX".SN50_N0017 )
      Coil( "00_Commissioning"."n0017-lv004-el001-k30001_SN50" )
   END_RUNG
   // the same network as SCL:
   "00_Commissioning"."n0017-lv004-el001-k30001_SN50" := "AlwaysTRUE" AND "ZAUX".SN50_N0017;
END_REGION

REGION Network 10: SN50_N0018
   RUNG wire#powerrail
      Contact( "AlwaysTRUE" )
      Contact( "ZAUX".SN50_N0018 )
      Coil( "00_Commissioning"."n0018-lv004-el001-k30001_SN50" )
   END_RUNG
   // the same network as SCL:
   "00_Commissioning"."n0018-lv004-el001-k30001_SN50" := "AlwaysTRUE" AND "ZAUX".SN50_N0018;
END_REGION

REGION Network 11: SN50_N0020
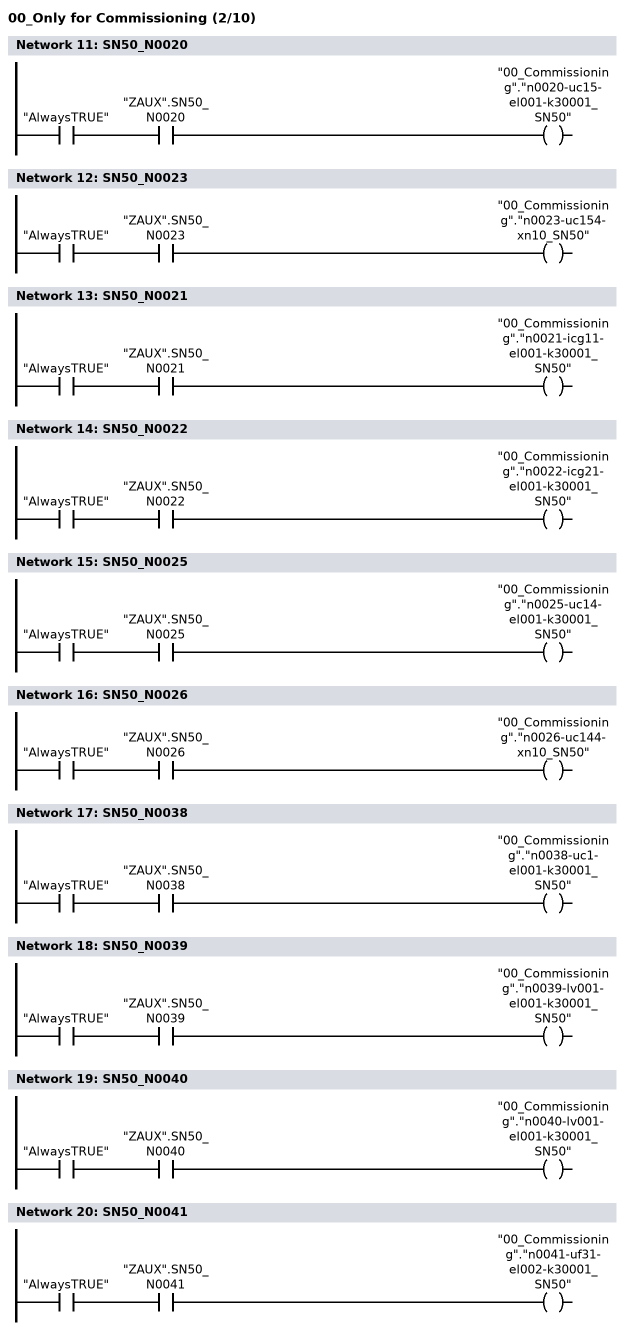
   RUNG wire#powerrail
      Contact( "AlwaysTRUE" )
      Contact( "ZAUX".SN50_N0020 )
      Coil( "00_Commissioning"."n0020-uc15-el001-k30001_SN50" )
   END_RUNG
   // the same network as SCL:
   "00_Commissioning"."n0020-uc15-el001-k30001_SN50" := "AlwaysTRUE" AND "ZAUX".SN50_N0020;
END_REGION

REGION Network 12: SN50_N0023
   RUNG wire#powerrail
      Contact( "AlwaysTRUE" )
      Contact( "ZAUX".SN50_N0023 )
      Coil( "00_Commissioning"."n0023-uc154-xn10_SN50" )
   END_RUNG
   // the same network as SCL:
   "00_Commissioning"."n0023-uc154-xn10_SN50" := "AlwaysTRUE" AND "ZAUX".SN50_N0023;
END_REGION

REGION Network 13: SN50_N0021
   RUNG wire#powerrail
      Contact( "AlwaysTRUE" )
      Contact( "ZAUX".SN50_N0021 )
      Coil( "00_Commissioning"."n0021-icg11-el001-k30001_SN50" )
   END_RUNG
   // the same network as SCL:
   "00_Commissioning"."n0021-icg11-el001-k30001_SN50" := "AlwaysTRUE" AND "ZAUX".SN50_N0021;
END_REGION

REGION Network 14: SN50_N0022
   RUNG wire#powerrail
      Contact( "AlwaysTRUE" )
      Contact( "ZAUX".SN50_N0022 )
      Coil( "00_Commissioning"."n0022-icg21-el001-k30001_SN50" )
   END_RUNG
   // the same network as SCL:
   "00_Commissioning"."n0022-icg21-el001-k30001_SN50" := "AlwaysTRUE" AND "ZAUX".SN50_N0022;
END_REGION

REGION Network 15: SN50_N0025
   RUNG wire#powerrail
      Contact( "AlwaysTRUE" )
      Contact( "ZAUX".SN50_N0025 )
      Coil( "00_Commissioning"."n0025-uc14-el001-k30001_SN50" )
   END_RUNG
   // the same network as SCL:
   "00_Commissioning"."n0025-uc14-el001-k30001_SN50" := "AlwaysTRUE" AND "ZAUX".SN50_N0025;
END_REGION

REGION Network 16: SN50_N0026
   RUNG wire#powerrail
      Contact( "AlwaysTRUE" )
      Contact( "ZAUX".SN50_N0026 )
      Coil( "00_Commissioning"."n0026-uc144-xn10_SN50" )
   END_RUNG
   // the same network as SCL:
   "00_Commissioning"."n0026-uc144-xn10_SN50" := "AlwaysTRUE" AND "ZAUX".SN50_N0026;
END_REGION

REGION Network 17: SN50_N0038
   RUNG wire#powerrail
      Contact( "AlwaysTRUE" )
      Contact( "ZAUX".SN50_N0038 )
      Coil( "00_Commissioning"."n0038-uc1-el001-k30001_SN50" )
   END_RUNG
   // the same network as SCL:
   "00_Commissioning"."n0038-uc1-el001-k30001_SN50" := "AlwaysTRUE" AND "ZAUX".SN50_N0038;
END_REGION

REGION Network 18: SN50_N0039
   RUNG wire#powerrail
      Contact( "AlwaysTRUE" )
      Contact( "ZAUX".SN50_N0039 )
      Coil( "00_Commissioning"."n0039-lv001-el001-k30001_SN50" )
   END_RUNG
   // the same network as SCL:
   "00_Commissioning"."n0039-lv001-el001-k30001_SN50" := "AlwaysTRUE" AND "ZAUX".SN50_N0039;
END_REGION

REGION Network 19: SN50_N0040
   RUNG wire#powerrail
      Contact( "AlwaysTRUE" )
      Contact( "ZAUX".SN50_N0040 )
      Coil( "00_Commissioning"."n0040-lv001-el001-k30001_SN50" )
   END_RUNG
   // the same network as SCL:
   "00_Commissioning"."n0040-lv001-el001-k30001_SN50" := "AlwaysTRUE" AND "ZAUX".SN50_N0040;
END_REGION

REGION Network 20: SN50_N0041
   RUNG wire#powerrail
      Contact( "AlwaysTRUE" )
      Contact( "ZAUX".SN50_N0041 )
      Coil( "00_Commissioning"."n0041-uf31-el002-k30001_SN50" )
   END_RUNG
   // the same network as SCL:
   "00_Commissioning"."n0041-uf31-el002-k30001_SN50" := "AlwaysTRUE" AND "ZAUX".SN50_N0041;
END_REGION

REGION Network 21: SN50_N0042
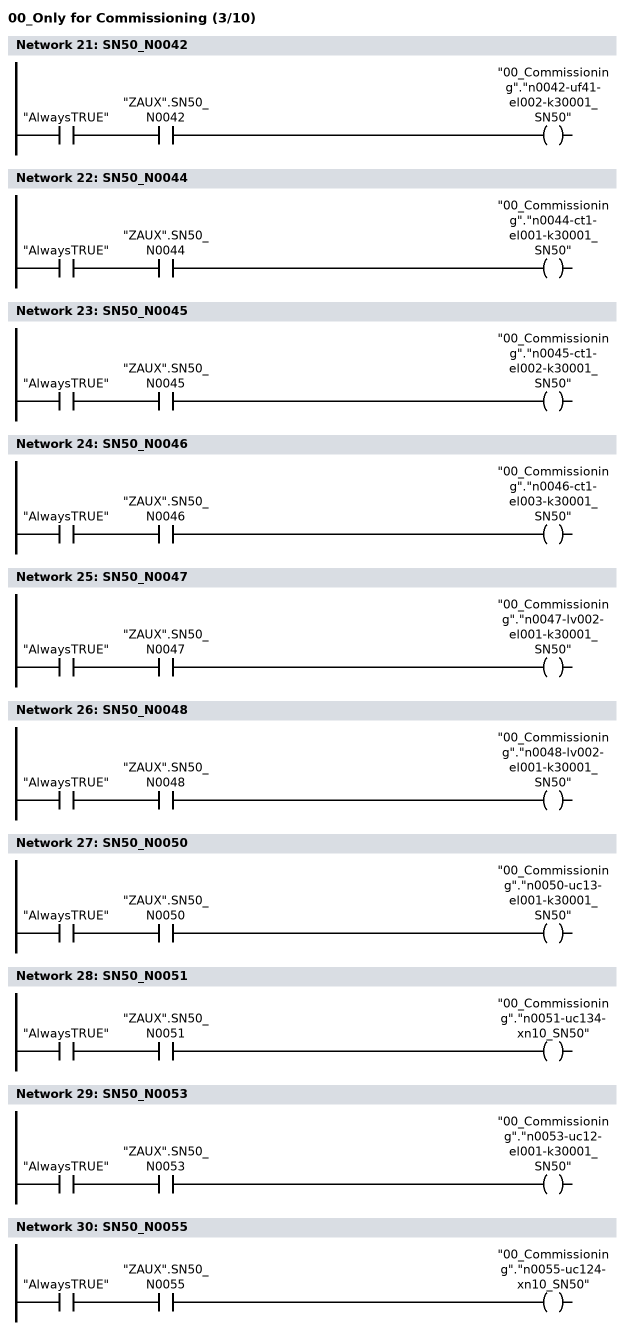
   RUNG wire#powerrail
      Contact( "AlwaysTRUE" )
      Contact( "ZAUX".SN50_N0042 )
      Coil( "00_Commissioning"."n0042-uf41-el002-k30001_SN50" )
   END_RUNG
   // the same network as SCL:
   "00_Commissioning"."n0042-uf41-el002-k30001_SN50" := "AlwaysTRUE" AND "ZAUX".SN50_N0042;
END_REGION

REGION Network 22: SN50_N0044
   RUNG wire#powerrail
      Contact( "AlwaysTRUE" )
      Contact( "ZAUX".SN50_N0044 )
      Coil( "00_Commissioning"."n0044-ct1-el001-k30001_SN50" )
   END_RUNG
   // the same network as SCL:
   "00_Commissioning"."n0044-ct1-el001-k30001_SN50" := "AlwaysTRUE" AND "ZAUX".SN50_N0044;
END_REGION

REGION Network 23: SN50_N0045
   RUNG wire#powerrail
      Contact( "AlwaysTRUE" )
      Contact( "ZAUX".SN50_N0045 )
      Coil( "00_Commissioning"."n0045-ct1-el002-k30001_SN50" )
   END_RUNG
   // the same network as SCL:
   "00_Commissioning"."n0045-ct1-el002-k30001_SN50" := "AlwaysTRUE" AND "ZAUX".SN50_N0045;
END_REGION

REGION Network 24: SN50_N0046
   RUNG wire#powerrail
      Contact( "AlwaysTRUE" )
      Contact( "ZAUX".SN50_N0046 )
      Coil( "00_Commissioning"."n0046-ct1-el003-k30001_SN50" )
   END_RUNG
   // the same network as SCL:
   "00_Commissioning"."n0046-ct1-el003-k30001_SN50" := "AlwaysTRUE" AND "ZAUX".SN50_N0046;
END_REGION

REGION Network 25: SN50_N0047
   RUNG wire#powerrail
      Contact( "AlwaysTRUE" )
      Contact( "ZAUX".SN50_N0047 )
      Coil( "00_Commissioning"."n0047-lv002-el001-k30001_SN50" )
   END_RUNG
   // the same network as SCL:
   "00_Commissioning"."n0047-lv002-el001-k30001_SN50" := "AlwaysTRUE" AND "ZAUX".SN50_N0047;
END_REGION

REGION Network 26: SN50_N0048
   RUNG wire#powerrail
      Contact( "AlwaysTRUE" )
      Contact( "ZAUX".SN50_N0048 )
      Coil( "00_Commissioning"."n0048-lv002-el001-k30001_SN50" )
   END_RUNG
   // the same network as SCL:
   "00_Commissioning"."n0048-lv002-el001-k30001_SN50" := "AlwaysTRUE" AND "ZAUX".SN50_N0048;
END_REGION

REGION Network 27: SN50_N0050
   RUNG wire#powerrail
      Contact( "AlwaysTRUE" )
      Contact( "ZAUX".SN50_N0050 )
      Coil( "00_Commissioning"."n0050-uc13-el001-k30001_SN50" )
   END_RUNG
   // the same network as SCL:
   "00_Commissioning"."n0050-uc13-el001-k30001_SN50" := "AlwaysTRUE" AND "ZAUX".SN50_N0050;
END_REGION

REGION Network 28: SN50_N0051
   RUNG wire#powerrail
      Contact( "AlwaysTRUE" )
      Contact( "ZAUX".SN50_N0051 )
      Coil( "00_Commissioning"."n0051-uc134-xn10_SN50" )
   END_RUNG
   // the same network as SCL:
   "00_Commissioning"."n0051-uc134-xn10_SN50" := "AlwaysTRUE" AND "ZAUX".SN50_N0051;
END_REGION

REGION Network 29: SN50_N0053
   RUNG wire#powerrail
      Contact( "AlwaysTRUE" )
      Contact( "ZAUX".SN50_N0053 )
      Coil( "00_Commissioning"."n0053-uc12-el001-k30001_SN50" )
   END_RUNG
   // the same network as SCL:
   "00_Commissioning"."n0053-uc12-el001-k30001_SN50" := "AlwaysTRUE" AND "ZAUX".SN50_N0053;
END_REGION

REGION Network 30: SN50_N0055
   RUNG wire#powerrail
      Contact( "AlwaysTRUE" )
      Contact( "ZAUX".SN50_N0055 )
      Coil( "00_Commissioning"."n0055-uc124-xn10_SN50" )
   END_RUNG
   // the same network as SCL:
   "00_Commissioning"."n0055-uc124-xn10_SN50" := "AlwaysTRUE" AND "ZAUX".SN50_N0055;
END_REGION

REGION Network 31: SN50_N0054
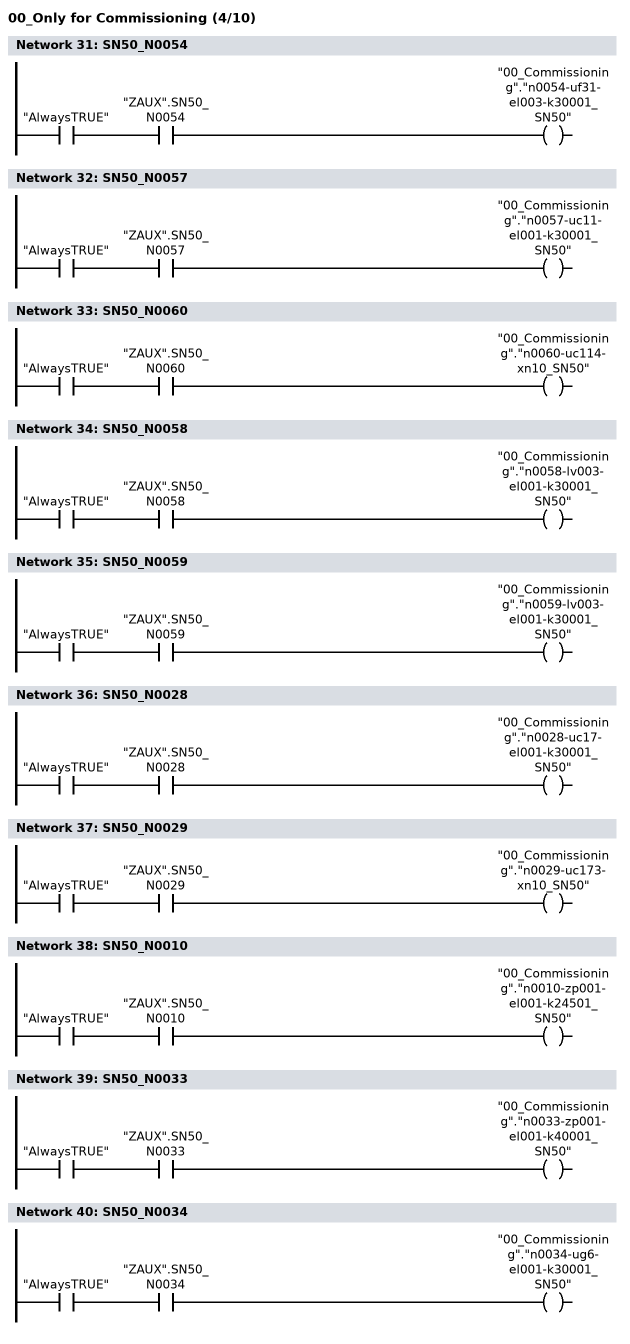
   RUNG wire#powerrail
      Contact( "AlwaysTRUE" )
      Contact( "ZAUX".SN50_N0054 )
      Coil( "00_Commissioning"."n0054-uf31-el003-k30001_SN50" )
   END_RUNG
   // the same network as SCL:
   "00_Commissioning"."n0054-uf31-el003-k30001_SN50" := "AlwaysTRUE" AND "ZAUX".SN50_N0054;
END_REGION

REGION Network 32: SN50_N0057
   RUNG wire#powerrail
      Contact( "AlwaysTRUE" )
      Contact( "ZAUX".SN50_N0057 )
      Coil( "00_Commissioning"."n0057-uc11-el001-k30001_SN50" )
   END_RUNG
   // the same network as SCL:
   "00_Commissioning"."n0057-uc11-el001-k30001_SN50" := "AlwaysTRUE" AND "ZAUX".SN50_N0057;
END_REGION

REGION Network 33: SN50_N0060
   RUNG wire#powerrail
      Contact( "AlwaysTRUE" )
      Contact( "ZAUX".SN50_N0060 )
      Coil( "00_Commissioning"."n0060-uc114-xn10_SN50" )
   END_RUNG
   // the same network as SCL:
   "00_Commissioning"."n0060-uc114-xn10_SN50" := "AlwaysTRUE" AND "ZAUX".SN50_N0060;
END_REGION

REGION Network 34: SN50_N0058
   RUNG wire#powerrail
      Contact( "AlwaysTRUE" )
      Contact( "ZAUX".SN50_N0058 )
      Coil( "00_Commissioning"."n0058-lv003-el001-k30001_SN50" )
   END_RUNG
   // the same network as SCL:
   "00_Commissioning"."n0058-lv003-el001-k30001_SN50" := "AlwaysTRUE" AND "ZAUX".SN50_N0058;
END_REGION

REGION Network 35: SN50_N0059
   RUNG wire#powerrail
      Contact( "AlwaysTRUE" )
      Contact( "ZAUX".SN50_N0059 )
      Coil( "00_Commissioning"."n0059-lv003-el001-k30001_SN50" )
   END_RUNG
   // the same network as SCL:
   "00_Commissioning"."n0059-lv003-el001-k30001_SN50" := "AlwaysTRUE" AND "ZAUX".SN50_N0059;
END_REGION

REGION Network 36: SN50_N0028
   RUNG wire#powerrail
      Contact( "AlwaysTRUE" )
      Contact( "ZAUX".SN50_N0028 )
      Coil( "00_Commissioning"."n0028-uc17-el001-k30001_SN50" )
   END_RUNG
   // the same network as SCL:
   "00_Commissioning"."n0028-uc17-el001-k30001_SN50" := "AlwaysTRUE" AND "ZAUX".SN50_N0028;
END_REGION

REGION Network 37: SN50_N0029
   RUNG wire#powerrail
      Contact( "AlwaysTRUE" )
      Contact( "ZAUX".SN50_N0029 )
      Coil( "00_Commissioning"."n0029-uc173-xn10_SN50" )
   END_RUNG
   // the same network as SCL:
   "00_Commissioning"."n0029-uc173-xn10_SN50" := "AlwaysTRUE" AND "ZAUX".SN50_N0029;
END_REGION

REGION Network 38: SN50_N0010
   RUNG wire#powerrail
      Contact( "AlwaysTRUE" )
      Contact( "ZAUX".SN50_N0010 )
      Coil( "00_Commissioning"."n0010-zp001-el001-k24501_SN50" )
   END_RUNG
   // the same network as SCL:
   "00_Commissioning"."n0010-zp001-el001-k24501_SN50" := "AlwaysTRUE" AND "ZAUX".SN50_N0010;
END_REGION

REGION Network 39: SN50_N0033
   RUNG wire#powerrail
      Contact( "AlwaysTRUE" )
      Contact( "ZAUX".SN50_N0033 )
      Coil( "00_Commissioning"."n0033-zp001-el001-k40001_SN50" )
   END_RUNG
   // the same network as SCL:
   "00_Commissioning"."n0033-zp001-el001-k40001_SN50" := "AlwaysTRUE" AND "ZAUX".SN50_N0033;
END_REGION

REGION Network 40: SN50_N0034
   RUNG wire#powerrail
      Contact( "AlwaysTRUE" )
      Contact( "ZAUX".SN50_N0034 )
      Coil( "00_Commissioning"."n0034-ug6-el001-k30001_SN50" )
   END_RUNG
   // the same network as SCL:
   "00_Commissioning"."n0034-ug6-el001-k30001_SN50" := "AlwaysTRUE" AND "ZAUX".SN50_N0034;
END_REGION

REGION Network 41: SN50_N0035
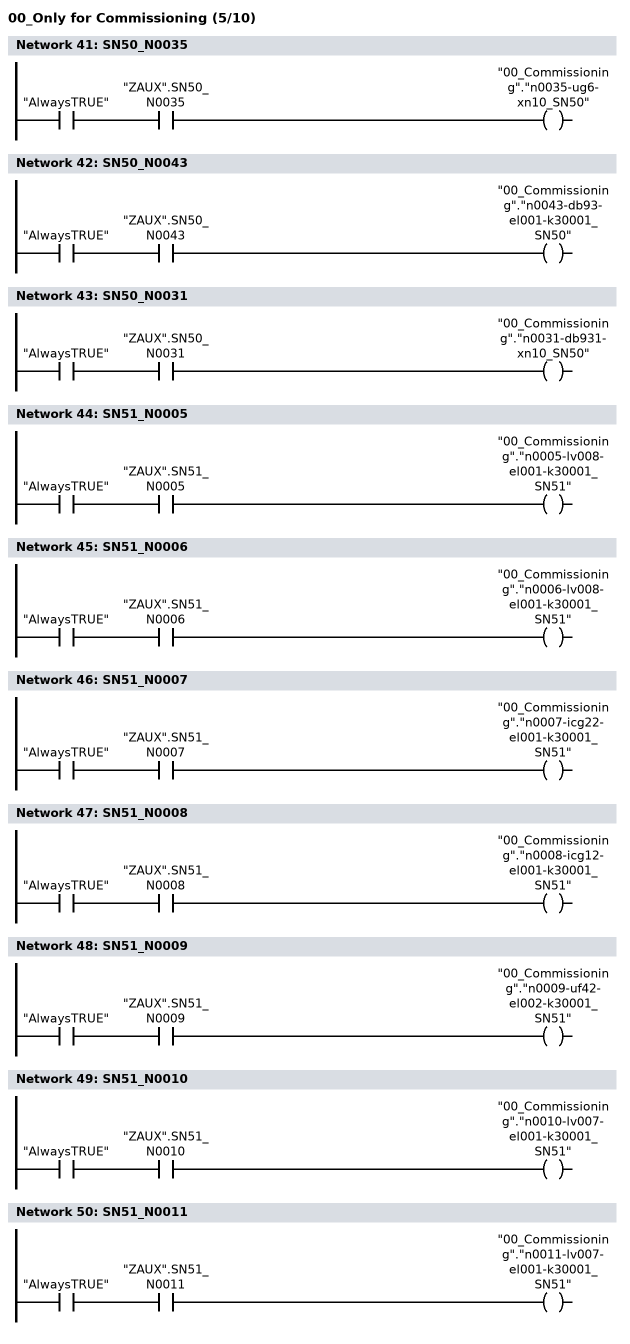
   RUNG wire#powerrail
      Contact( "AlwaysTRUE" )
      Contact( "ZAUX".SN50_N0035 )
      Coil( "00_Commissioning"."n0035-ug6-xn10_SN50" )
   END_RUNG
   // the same network as SCL:
   "00_Commissioning"."n0035-ug6-xn10_SN50" := "AlwaysTRUE" AND "ZAUX".SN50_N0035;
END_REGION

REGION Network 42: SN50_N0043
   RUNG wire#powerrail
      Contact( "AlwaysTRUE" )
      Contact( "ZAUX".SN50_N0043 )
      Coil( "00_Commissioning"."n0043-db93-el001-k30001_SN50" )
   END_RUNG
   // the same network as SCL:
   "00_Commissioning"."n0043-db93-el001-k30001_SN50" := "AlwaysTRUE" AND "ZAUX".SN50_N0043;
END_REGION

REGION Network 43: SN50_N0031
   RUNG wire#powerrail
      Contact( "AlwaysTRUE" )
      Contact( "ZAUX".SN50_N0031 )
      Coil( "00_Commissioning"."n0031-db931-xn10_SN50" )
   END_RUNG
   // the same network as SCL:
   "00_Commissioning"."n0031-db931-xn10_SN50" := "AlwaysTRUE" AND "ZAUX".SN50_N0031;
END_REGION

REGION Network 44: SN51_N0005
   RUNG wire#powerrail
      Contact( "AlwaysTRUE" )
      Contact( "ZAUX".SN51_N0005 )
      Coil( "00_Commissioning"."n0005-lv008-el001-k30001_SN51" )
   END_RUNG
   // the same network as SCL:
   "00_Commissioning"."n0005-lv008-el001-k30001_SN51" := "AlwaysTRUE" AND "ZAUX".SN51_N0005;
END_REGION

REGION Network 45: SN51_N0006
   RUNG wire#powerrail
      Contact( "AlwaysTRUE" )
      Contact( "ZAUX".SN51_N0006 )
      Coil( "00_Commissioning"."n0006-lv008-el001-k30001_SN51" )
   END_RUNG
   // the same network as SCL:
   "00_Commissioning"."n0006-lv008-el001-k30001_SN51" := "AlwaysTRUE" AND "ZAUX".SN51_N0006;
END_REGION

REGION Network 46: SN51_N0007
   RUNG wire#powerrail
      Contact( "AlwaysTRUE" )
      Contact( "ZAUX".SN51_N0007 )
      Coil( "00_Commissioning"."n0007-icg22-el001-k30001_SN51" )
   END_RUNG
   // the same network as SCL:
   "00_Commissioning"."n0007-icg22-el001-k30001_SN51" := "AlwaysTRUE" AND "ZAUX".SN51_N0007;
END_REGION

REGION Network 47: SN51_N0008
   RUNG wire#powerrail
      Contact( "AlwaysTRUE" )
      Contact( "ZAUX".SN51_N0008 )
      Coil( "00_Commissioning"."n0008-icg12-el001-k30001_SN51" )
   END_RUNG
   // the same network as SCL:
   "00_Commissioning"."n0008-icg12-el001-k30001_SN51" := "AlwaysTRUE" AND "ZAUX".SN51_N0008;
END_REGION

REGION Network 48: SN51_N0009
   RUNG wire#powerrail
      Contact( "AlwaysTRUE" )
      Contact( "ZAUX".SN51_N0009 )
      Coil( "00_Commissioning"."n0009-uf42-el002-k30001_SN51" )
   END_RUNG
   // the same network as SCL:
   "00_Commissioning"."n0009-uf42-el002-k30001_SN51" := "AlwaysTRUE" AND "ZAUX".SN51_N0009;
END_REGION

REGION Network 49: SN51_N0010
   RUNG wire#powerrail
      Contact( "AlwaysTRUE" )
      Contact( "ZAUX".SN51_N0010 )
      Coil( "00_Commissioning"."n0010-lv007-el001-k30001_SN51" )
   END_RUNG
   // the same network as SCL:
   "00_Commissioning"."n0010-lv007-el001-k30001_SN51" := "AlwaysTRUE" AND "ZAUX".SN51_N0010;
END_REGION

REGION Network 50: SN51_N0011
   RUNG wire#powerrail
      Contact( "AlwaysTRUE" )
      Contact( "ZAUX".SN51_N0011 )
      Coil( "00_Commissioning"."n0011-lv007-el001-k30001_SN51" )
   END_RUNG
   // the same network as SCL:
   "00_Commissioning"."n0011-lv007-el001-k30001_SN51" := "AlwaysTRUE" AND "ZAUX".SN51_N0011;
END_REGION

REGION Network 51: SN51_N0021
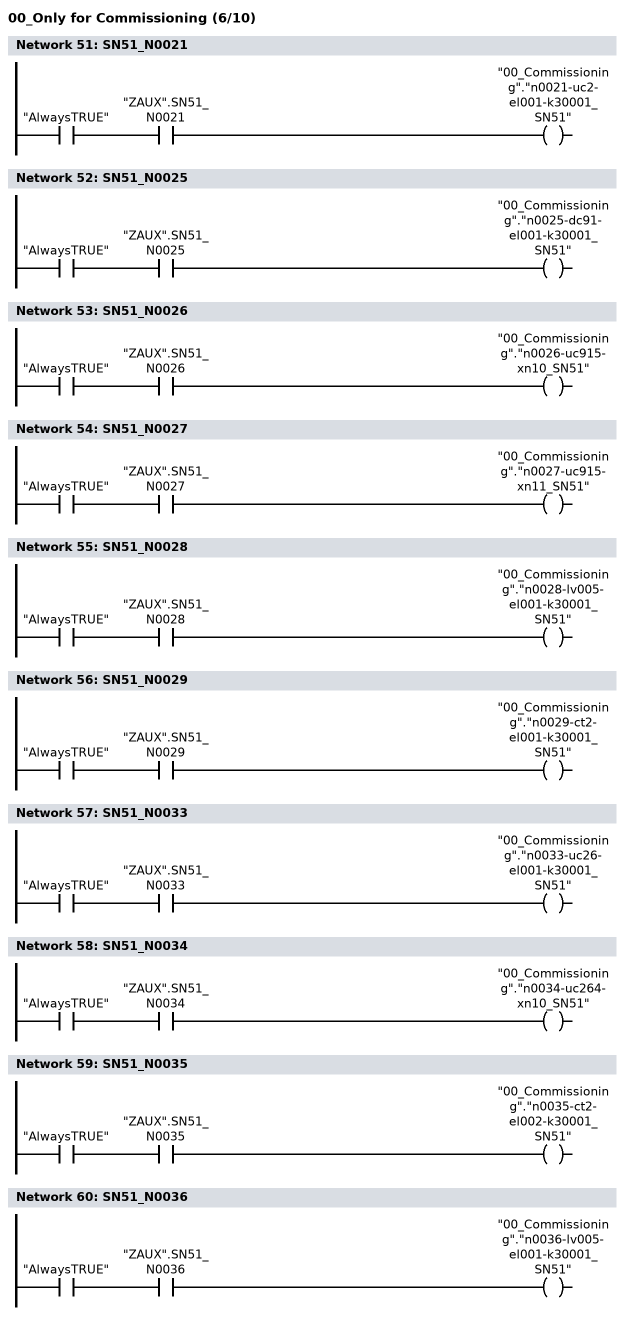
   RUNG wire#powerrail
      Contact( "AlwaysTRUE" )
      Contact( "ZAUX".SN51_N0021 )
      Coil( "00_Commissioning"."n0021-uc2-el001-k30001_SN51" )
   END_RUNG
   // the same network as SCL:
   "00_Commissioning"."n0021-uc2-el001-k30001_SN51" := "AlwaysTRUE" AND "ZAUX".SN51_N0021;
END_REGION

REGION Network 52: SN51_N0025
   RUNG wire#powerrail
      Contact( "AlwaysTRUE" )
      Contact( "ZAUX".SN51_N0025 )
      Coil( "00_Commissioning"."n0025-dc91-el001-k30001_SN51" )
   END_RUNG
   // the same network as SCL:
   "00_Commissioning"."n0025-dc91-el001-k30001_SN51" := "AlwaysTRUE" AND "ZAUX".SN51_N0025;
END_REGION

REGION Network 53: SN51_N0026
   RUNG wire#powerrail
      Contact( "AlwaysTRUE" )
      Contact( "ZAUX".SN51_N0026 )
      Coil( "00_Commissioning"."n0026-uc915-xn10_SN51" )
   END_RUNG
   // the same network as SCL:
   "00_Commissioning"."n0026-uc915-xn10_SN51" := "AlwaysTRUE" AND "ZAUX".SN51_N0026;
END_REGION

REGION Network 54: SN51_N0027
   RUNG wire#powerrail
      Contact( "AlwaysTRUE" )
      Contact( "ZAUX".SN51_N0027 )
      Coil( "00_Commissioning"."n0027-uc915-xn11_SN51" )
   END_RUNG
   // the same network as SCL:
   "00_Commissioning"."n0027-uc915-xn11_SN51" := "AlwaysTRUE" AND "ZAUX".SN51_N0027;
END_REGION

REGION Network 55: SN51_N0028
   RUNG wire#powerrail
      Contact( "AlwaysTRUE" )
      Contact( "ZAUX".SN51_N0028 )
      Coil( "00_Commissioning"."n0028-lv005-el001-k30001_SN51" )
   END_RUNG
   // the same network as SCL:
   "00_Commissioning"."n0028-lv005-el001-k30001_SN51" := "AlwaysTRUE" AND "ZAUX".SN51_N0028;
END_REGION

REGION Network 56: SN51_N0029
   RUNG wire#powerrail
      Contact( "AlwaysTRUE" )
      Contact( "ZAUX".SN51_N0029 )
      Coil( "00_Commissioning"."n0029-ct2-el001-k30001_SN51" )
   END_RUNG
   // the same network as SCL:
   "00_Commissioning"."n0029-ct2-el001-k30001_SN51" := "AlwaysTRUE" AND "ZAUX".SN51_N0029;
END_REGION

REGION Network 57: SN51_N0033
   RUNG wire#powerrail
      Contact( "AlwaysTRUE" )
      Contact( "ZAUX".SN51_N0033 )
      Coil( "00_Commissioning"."n0033-uc26-el001-k30001_SN51" )
   END_RUNG
   // the same network as SCL:
   "00_Commissioning"."n0033-uc26-el001-k30001_SN51" := "AlwaysTRUE" AND "ZAUX".SN51_N0033;
END_REGION

REGION Network 58: SN51_N0034
   RUNG wire#powerrail
      Contact( "AlwaysTRUE" )
      Contact( "ZAUX".SN51_N0034 )
      Coil( "00_Commissioning"."n0034-uc264-xn10_SN51" )
   END_RUNG
   // the same network as SCL:
   "00_Commissioning"."n0034-uc264-xn10_SN51" := "AlwaysTRUE" AND "ZAUX".SN51_N0034;
END_REGION

REGION Network 59: SN51_N0035
   RUNG wire#powerrail
      Contact( "AlwaysTRUE" )
      Contact( "ZAUX".SN51_N0035 )
      Coil( "00_Commissioning"."n0035-ct2-el002-k30001_SN51" )
   END_RUNG
   // the same network as SCL:
   "00_Commissioning"."n0035-ct2-el002-k30001_SN51" := "AlwaysTRUE" AND "ZAUX".SN51_N0035;
END_REGION

REGION Network 60: SN51_N0036
   RUNG wire#powerrail
      Contact( "AlwaysTRUE" )
      Contact( "ZAUX".SN51_N0036 )
      Coil( "00_Commissioning"."n0036-lv005-el001-k30001_SN51" )
   END_RUNG
   // the same network as SCL:
   "00_Commissioning"."n0036-lv005-el001-k30001_SN51" := "AlwaysTRUE" AND "ZAUX".SN51_N0036;
END_REGION

REGION Network 61: SN51_N0041
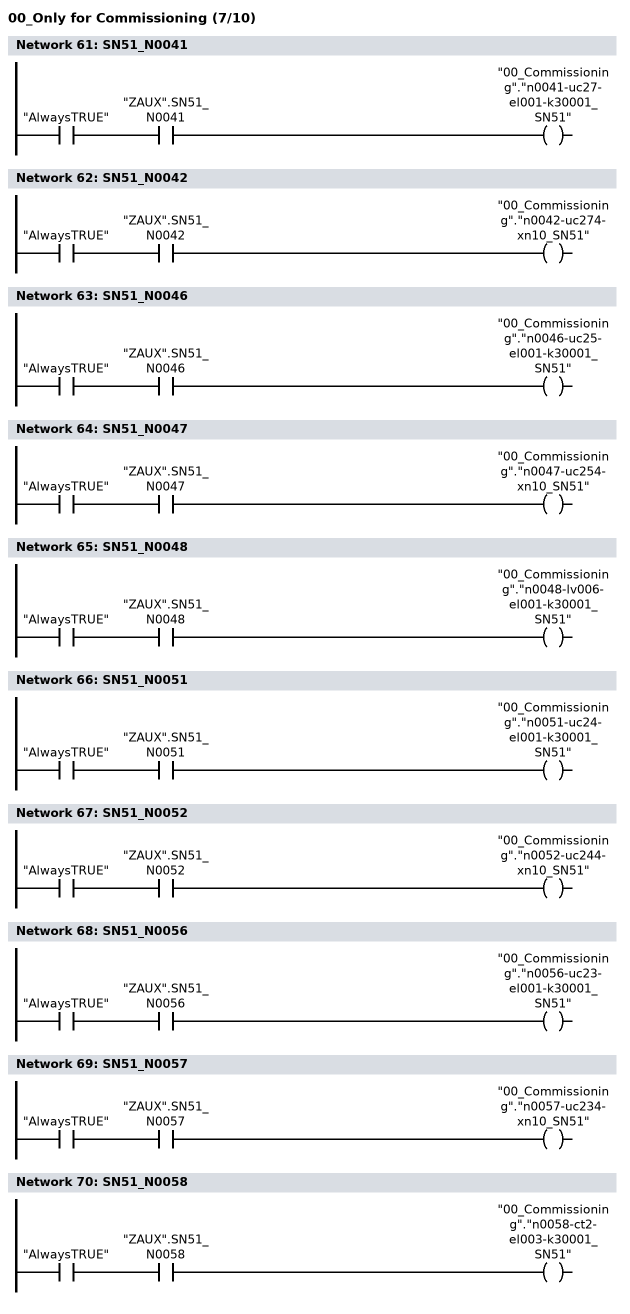
   RUNG wire#powerrail
      Contact( "AlwaysTRUE" )
      Contact( "ZAUX".SN51_N0041 )
      Coil( "00_Commissioning"."n0041-uc27-el001-k30001_SN51" )
   END_RUNG
   // the same network as SCL:
   "00_Commissioning"."n0041-uc27-el001-k30001_SN51" := "AlwaysTRUE" AND "ZAUX".SN51_N0041;
END_REGION

REGION Network 62: SN51_N0042
   RUNG wire#powerrail
      Contact( "AlwaysTRUE" )
      Contact( "ZAUX".SN51_N0042 )
      Coil( "00_Commissioning"."n0042-uc274-xn10_SN51" )
   END_RUNG
   // the same network as SCL:
   "00_Commissioning"."n0042-uc274-xn10_SN51" := "AlwaysTRUE" AND "ZAUX".SN51_N0042;
END_REGION

REGION Network 63: SN51_N0046
   RUNG wire#powerrail
      Contact( "AlwaysTRUE" )
      Contact( "ZAUX".SN51_N0046 )
      Coil( "00_Commissioning"."n0046-uc25-el001-k30001_SN51" )
   END_RUNG
   // the same network as SCL:
   "00_Commissioning"."n0046-uc25-el001-k30001_SN51" := "AlwaysTRUE" AND "ZAUX".SN51_N0046;
END_REGION

REGION Network 64: SN51_N0047
   RUNG wire#powerrail
      Contact( "AlwaysTRUE" )
      Contact( "ZAUX".SN51_N0047 )
      Coil( "00_Commissioning"."n0047-uc254-xn10_SN51" )
   END_RUNG
   // the same network as SCL:
   "00_Commissioning"."n0047-uc254-xn10_SN51" := "AlwaysTRUE" AND "ZAUX".SN51_N0047;
END_REGION

REGION Network 65: SN51_N0048
   RUNG wire#powerrail
      Contact( "AlwaysTRUE" )
      Contact( "ZAUX".SN51_N0048 )
      Coil( "00_Commissioning"."n0048-lv006-el001-k30001_SN51" )
   END_RUNG
   // the same network as SCL:
   "00_Commissioning"."n0048-lv006-el001-k30001_SN51" := "AlwaysTRUE" AND "ZAUX".SN51_N0048;
END_REGION

REGION Network 66: SN51_N0051
   RUNG wire#powerrail
      Contact( "AlwaysTRUE" )
      Contact( "ZAUX".SN51_N0051 )
      Coil( "00_Commissioning"."n0051-uc24-el001-k30001_SN51" )
   END_RUNG
   // the same network as SCL:
   "00_Commissioning"."n0051-uc24-el001-k30001_SN51" := "AlwaysTRUE" AND "ZAUX".SN51_N0051;
END_REGION

REGION Network 67: SN51_N0052
   RUNG wire#powerrail
      Contact( "AlwaysTRUE" )
      Contact( "ZAUX".SN51_N0052 )
      Coil( "00_Commissioning"."n0052-uc244-xn10_SN51" )
   END_RUNG
   // the same network as SCL:
   "00_Commissioning"."n0052-uc244-xn10_SN51" := "AlwaysTRUE" AND "ZAUX".SN51_N0052;
END_REGION

REGION Network 68: SN51_N0056
   RUNG wire#powerrail
      Contact( "AlwaysTRUE" )
      Contact( "ZAUX".SN51_N0056 )
      Coil( "00_Commissioning"."n0056-uc23-el001-k30001_SN51" )
   END_RUNG
   // the same network as SCL:
   "00_Commissioning"."n0056-uc23-el001-k30001_SN51" := "AlwaysTRUE" AND "ZAUX".SN51_N0056;
END_REGION

REGION Network 69: SN51_N0057
   RUNG wire#powerrail
      Contact( "AlwaysTRUE" )
      Contact( "ZAUX".SN51_N0057 )
      Coil( "00_Commissioning"."n0057-uc234-xn10_SN51" )
   END_RUNG
   // the same network as SCL:
   "00_Commissioning"."n0057-uc234-xn10_SN51" := "AlwaysTRUE" AND "ZAUX".SN51_N0057;
END_REGION

REGION Network 70: SN51_N0058
   RUNG wire#powerrail
      Contact( "AlwaysTRUE" )
      Contact( "ZAUX".SN51_N0058 )
      Coil( "00_Commissioning"."n0058-ct2-el003-k30001_SN51" )
   END_RUNG
   // the same network as SCL:
   "00_Commissioning"."n0058-ct2-el003-k30001_SN51" := "AlwaysTRUE" AND "ZAUX".SN51_N0058;
END_REGION

REGION Network 71: SN51_N0061
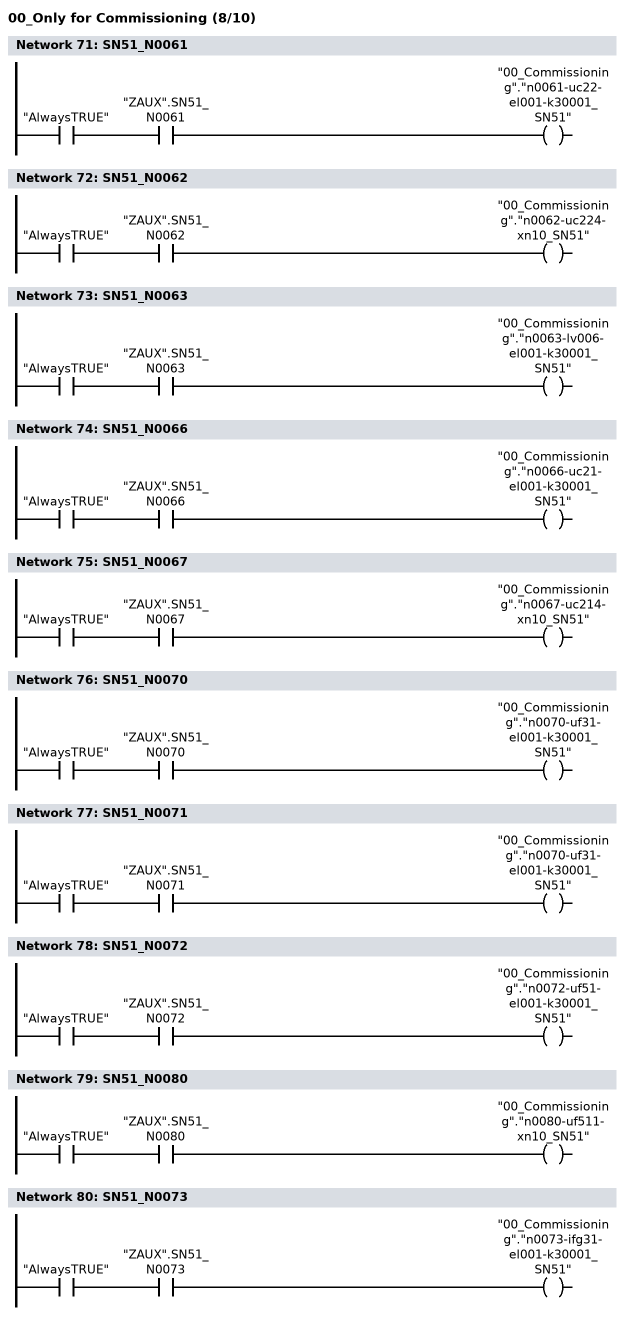
   RUNG wire#powerrail
      Contact( "AlwaysTRUE" )
      Contact( "ZAUX".SN51_N0061 )
      Coil( "00_Commissioning"."n0061-uc22-el001-k30001_SN51" )
   END_RUNG
   // the same network as SCL:
   "00_Commissioning"."n0061-uc22-el001-k30001_SN51" := "AlwaysTRUE" AND "ZAUX".SN51_N0061;
END_REGION

REGION Network 72: SN51_N0062
   RUNG wire#powerrail
      Contact( "AlwaysTRUE" )
      Contact( "ZAUX".SN51_N0062 )
      Coil( "00_Commissioning"."n0062-uc224-xn10_SN51" )
   END_RUNG
   // the same network as SCL:
   "00_Commissioning"."n0062-uc224-xn10_SN51" := "AlwaysTRUE" AND "ZAUX".SN51_N0062;
END_REGION

